C01835=1198.464,47.154,-46.353,-179.303,5.739,148.808
C01836=1198.459,47.403,-46.370,-179.300,5.741,148.808
C01837=1198.454,47.653,-46.386,-179.297,5.741,148.807
C01838=1198.449,47.901,-46.402,-179.295,5.742,148.806
C01839=1198.445,48.152,-46.418,-179.292,5.743,148.806
C01840=1198.439,48.401,-46.434,-179.290,5.743,148.805
C01841=1198.435,48.650,-46.450,-179.287,5.744,148.804
C01842=1198.429,48.900,-46.466,-179.284,5.744,148.804
C01843=1198.425,49.149,-46.482,-179.282,5.745,148.803
C01844=1198.419,49.399,-46.498,-179.280,5.746,148.803
C01845=1198.414,49.647,-46.514,-179.276,5.747,148.802
C01846=1198.410,49.898,-46.530,-179.274,5.748,148.801
C01847=1198.404,50.146,-46.547,-179.272,5.749,148.801
C01848=1198.400,50.396,-46.563,-179.269,5.749,148.800
C01849=1198.395,50.645,-46.579,-179.266,5.750,148.800
C01850=1198.390,50.895,-46.595,-179.264,5.751,148.799
C01851=1198.385,51.144,-46.611,-179.262,5.751,148.798
C01852=1198.380,51.394,-46.627,-179.258,5.753,148.798
C01853=1198.375,51.643,-46.643,-179.256,5.753,148.797
C01854=1198.370,51.893,-46.659,-179.254,5.754,148.797
C01855=1198.365,52.142,-46.676,-179.251,5.754,148.796
C01856=1198.360,52.391,-46.692,-179.248,5.755,148.795
C01857=1198.355,52.641,-46.708,-179.246,5.756,148.795
C01858=1198.351,52.890,-46.725,-179.244,5.756,148.794
C01859=1198.345,53.140,-46.740,-179.240,5.758,148.794
C01860=1198.341,53.389,-46.757,-179.238,5.759,148.793
C01861=1198.336,53.638,-46.773,-179.236,5.759,148.792
C01862=1198.331,53.888,-46.789,-179.233,5.760,148.792
C01863=1198.326,54.138,-46.806,-179.231,5.761,148.791
C01864=1198.321,54.387,-46.823,-179.228,5.761,148.791
C01865=1198.315,54.655,-46.840,-179.225,5.763,148.790
C01866=1198.310,54.924,-46.857,-179.222,5.763,148.789
C01867=1198.305,55.192,-46.875,-179.220,5.764,148.789
C01868=1198.299,55.461,-46.892,-179.216,5.765,148.788
C01869=1198.294,55.710,-46.909,-179.214,5.766,148.788
C01870=1198.290,55.960,-46.926,-179.212,5.766,148.787
C01871=1198.284,56.209,-46.941,-179.209,5.767,148.786
C01872=1198.280,56.459,-46.958,-179.207,5.768,148.786
C01873=1198.275,56.708,-46.974,-179.204,5.768,148.785
C01874=1198.270,56.957,-46.991,-179.201,5.770,148.784
C01875=1198.264,57.207,-47.007,-179.199,5.771,148.784
C01876=1198.260,57.456,-47.024,-179.196,5.771,148.783
C01877=1198.255,57.706,-47.040,-179.194,5.772,148.783
C01878=1198.250,57.955,-47.057,-179.191,5.772,148.782
C01879=1198.244,58.205,-47.073,-179.189,5.773,148.782
C01880=1198.239,58.454,-47.090,-179.186,5.775,148.781
C01881=1198.235,58.703,-47.106,-179.183,5.775,148.780
C01882=1198.230,58.953,-47.123,-179.181,5.776,148.780
C01883=1198.225,59.201,-47.139,-179.178,5.777,148.779
C01884=1198.220,59.452,-47.156,-179.176,5.777,148.779
C01885=1198.215,59.701,-47.172,-179.173,5.778,148.778
C01886=1198.210,59.950,-47.189,-179.170,5.779,148.777
C01887=1198.206,60.200,-47.205,-179.168,5.780,148.777
C01888=1198.200,60.449,-47.222,-179.165,5.781,148.776
C01889=1198.195,60.698,-47.239,-179.163,5.781,148.776
C01890=1198.191,60.948,-47.256,-179.160,5.782,148.775
C01891=1198.185,61.197,-47.273,-179.157,5.784,148.775
C01892=1198.180,61.447,-47.289,-179.155,5.784,148.774
C01893=1198.176,61.696,-47.305,-179.152,5.785,148.773
C01894=1198.171,61.945,-47.321,-179.150,5.786,148.773
C01895=1198.166,62.195,-47.339,-179.147,5.786,148.772
C01896=1198.161,62.444,-47.355,-179.144,5.787,148.771
C01897=1198.156,62.693,-47.372,-179.142,5.788,148.771
C01898=1198.151,62.943,-47.389,-179.139,5.789,148.770
C01899=1198.146,63.192,-47.406,-179.137,5.789,148.770
C01900=1198.141,63.441,-47.422,-179.135,5.790,148.769
C01901=1198.136,63.691,-47.439,-179.131,5.792,148.769
C01902=1198.132,63.941,-47.456,-179.129,5.792,148.768
C01903=1198.126,64.189,-47.472,-179.127,5.793,148.768
C01904=1198.121,64.439,-47.489,-179.124,5.794,148.767
C01905=1198.117,64.689,-47.506,-179.122,5.795,148.766
C01906=1198.112,64.938,-47.523,-179.119,5.796,148.766
C01907=1198.106,65.187,-47.540,-179.116,5.796,148.765
C01908=1198.102,65.437,-47.556,-179.114,5.797,148.765
C01909=1198.097,65.686,-47.574,-179.111,5.798,148.764
C01910=1198.092,65.935,-47.590,-179.109,5.798,148.763
C01911=1198.086,66.185,-47.607,-179.106,5.800,148.763
C01912=1198.082,66.435,-47.624,-179.103,5.801,148.762
C01913=1198.078,66.684,-47.641,-179.101,5.801,148.762
C01914=1198.072,66.933,-47.657,-179.099,5.802,148.761
C01915=1198.067,67.183,-47.674,-179.095,5.804,148.760
C01916=1198.062,67.432,-47.692,-179.093,5.804,148.760
C01917=1198.058,67.681,-47.709,-179.091,5.805,148.759
C01918=1198.052,67.930,-47.726,-179.088,5.806,148.759
C01919=1198.048,68.180,-47.742,-179.085,5.806,148.758
C01920=1198.043,68.429,-47.759,-179.083,5.808,148.758
C01921=1198.038,68.679,-47.776,-179.080,5.808,148.757
C01922=1198.033,68.929,-47.793,-179.078,5.809,148.757
C01923=1198.028,69.177,-47.811,-179.075,5.810,148.756
C01924=1198.023,69.427,-47.827,-179.072,5.811,148.755
C01925=1198.018,69.676,-47.844,-179.070,5.812,148.755
C01926=1198.014,69.926,-47.861,-179.067,5.813,148.754
C01927=1198.008,70.176,-47.878,-179.065,5.813,148.753
C01928=1198.004,70.424,-47.895,-179.062,5.815,148.753
C01929=1197.998,70.674,-47.913,-179.059,5.815,148.752
C01930=1197.994,70.923,-47.929,-179.057,5.816,148.752
C01931=1197.989,71.173,-47.947,-179.054,5.817,148.751
C01932=1197.984,71.422,-47.965,-179.051,5.818,148.751
C01933=1197.979,71.671,-47.981,-179.049,5.819,148.750
C01934=1197.974,71.921,-47.998,-179.046,5.820,148.750
C01935=1197.969,72.170,-48.015,-179.044,5.820,148.749
C01936=1197.964,72.419,-48.033,-179.041,5.822,148.748
C01937=1197.960,72.669,-48.050,-179.038,5.823,148.748
C01938=1197.954,72.919,-48.067,-179.036,5.824,148.747
C01939=1197.949,73.167,-48.084,-179.034,5.824,148.747
C01940=1197.944,73.417,-48.101,-179.030,5.825,148.746
C01941=1197.939,73.666,-48.118,-179.028,5.826,148.746
C01942=1197.935,73.915,-48.136,-179.026,5.827,148.745
C01943=1197.930,74.165,-48.153,-179.023,5.827,148.744
C01944=1197.925,74.415,-48.170,-179.020,5.829,148.744
C01945=1197.920,74.664,-48.188,-179.018,5.830,148.743
C01946=1197.915,74.913,-48.205,-179.016,5.831,148.743
C01947=1197.910,75.162,-48.222,-179.013,5.831,148.742
C01948=1197.905,75.411,-48.239,-179.010,5.833,148.742
C01949=1197.900,75.661,-48.256,-179.008,5.833,148.741
C01950=1197.896,75.910,-48.274,-179.005,5.834,148.740
C01951=1197.891,76.160,-48.291,-179.002,5.836,148.740
C01952=1197.886,76.409,-48.309,-179.000,5.836,148.739
C01953=1197.881,76.659,-48.326,-178.997,5.837,148.739
C01954=1197.876,76.908,-48.344,-178.995,5.838,148.738
C01955=1197.871,77.157,-48.361,-178.992,5.839,148.738
C01956=1197.866,77.406,-48.378,-178.990,5.840,148.737
C01957=1197.861,77.655,-48.395,-178.987,5.841,148.737
C01958=1197.856,77.905,-48.413,-178.984,5.841,148.736
C01959=1197.851,78.154,-48.430,-178.982,5.843,148.735
C01960=1197.847,78.403,-48.448,-178.979,5.843,148.735
C01961=1197.842,78.653,-48.465,-178.977,5.844,148.734
C01962=1197.837,78.902,-48.483,-178.974,5.846,148.734
C01963=1197.831,79.152,-48.500,-178.971,5.846,148.733
C01964=1197.827,79.401,-48.518,-178.969,5.847,148.733
C01965=1197.822,79.651,-48.535,-178.966,5.849,148.732
C01966=1197.817,79.900,-48.553,-178.964,5.850,148.732
C01967=1197.812,80.150,-48.570,-178.961,5.850,148.731
C01968=1197.808,80.399,-48.588,-178.958,5.851,148.730
C01969=1197.802,80.667,-48.606,-178.956,5.852,148.730
C01970=1197.797,80.935,-48.625,-178.953,5.853,148.729
C01971=1197.791,81.204,-48.644,-178.950,5.854,148.729
C01972=1197.786,81.472,-48.664,-178.947,5.855,148.728
C01973=1197.781,81.721,-48.681,-178.944,5.857,148.727
C01974=1197.777,81.971,-48.698,-178.942,5.857,148.727
C01975=1197.772,82.220,-48.716,-178.940,5.858,148.726
C01976=1197.767,82.469,-48.734,-178.936,5.859,148.726
C01977=1197.762,82.719,-48.751,-178.934,5.860,148.725
C01978=1197.757,82.968,-48.769,-178.932,5.861,148.725
C01979=1197.752,83.217,-48.787,-178.928,5.862,148.724
C01980=1197.747,83.467,-48.804,-178.926,5.863,148.724
C01981=1197.743,83.716,-48.822,-178.924,5.864,148.723
C01982=1197.738,83.965,-48.840,-178.921,5.864,148.722
C01983=1197.732,84.215,-48.857,-178.918,5.866,148.722
C01984=1197.728,84.464,-48.875,-178.916,5.867,148.721
C01985=1197.723,84.713,-48.893,-178.914,5.868,148.721
C01986=1197.718,84.962,-48.911,-178.910,5.869,148.720
C01987=1197.713,85.212,-48.928,-178.908,5.870,148.720
C01988=1197.708,85.461,-48.946,-178.906,5.870,148.719
C01989=1197.703,85.710,-48.964,-178.903,5.872,148.719
C01990=1197.699,85.959,-48.982,-178.900,5.873,148.718
C01991=1197.694,86.209,-49.000,-178.898,5.873,148.717
C01992=1197.688,86.458,-49.017,-178.895,5.875,148.717
C01993=1197.683,86.708,-49.035,-178.892,5.876,148.716
C01994=1197.679,86.957,-49.053,-178.890,5.876,148.716
C01995=1197.674,87.207,-49.071,-178.887,5.878,148.715
C01996=1197.669,87.456,-49.089,-178.885,5.879,148.715
C01997=1197.664,87.705,-49.107,-178.882,5.879,148.714
C01998=1197.659,87.955,-49.125,-178.879,5.881,148.713
C01999=1197.654,88.204,-49.143,-178.877,5.882,148.713
C02000=1197.649,88.453,-49.161,-178.874,5.883,148.712
C02001=1197.644,88.702,-49.178,-178.872,5.884,148.712
C02002=1197.640,88.951,-49.196,-178.869,5.884,148.711
C02003=1197.635,89.201,-49.214,-178.866,5.886,148.711
C02004=1197.630,89.451,-49.233,-178.864,5.887,148.710
C02005=1197.625,89.700,-49.251,-178.861,5.888,148.710
C02006=1197.621,89.949,-49.269,-178.858,5.889,148.709
C02007=1197.616,90.198,-49.287,-178.856,5.890,148.709
C02008=1197.611,90.447,-49.305,-178.854,5.891,148.708
C02009=1197.606,90.696,-49.323,-178.850,5.892,148.707
C02010=1197.601,90.946,-49.341,-178.848,5.893,148.707
C02011=1197.596,91.195,-49.359,-178.846,5.893,148.706
C02012=1197.592,91.445,-49.377,-178.843,5.895,148.706
C02013=1197.587,91.694,-49.395,-178.840,5.896,148.705
C02014=1197.582,91.943,-49.413,-178.838,5.898,148.705
C02015=1197.577,92.192,-49.431,-178.835,5.898,148.704
C02016=1197.572,92.441,-49.449,-178.833,5.899,148.704
C02017=1197.567,92.690,-49.467,-178.830,5.900,148.703
C02018=1197.562,92.941,-49.486,-178.827,5.901,148.703
C02019=1197.557,93.190,-49.504,-178.825,5.902,148.702
C02020=1197.552,93.439,-49.522,-178.822,5.904,148.702
C02021=1197.547,93.688,-49.540,-178.820,5.904,148.701
C02022=1197.542,93.937,-49.558,-178.817,5.906,148.701
C02023=1197.538,94.187,-49.576,-178.814,5.906,148.700
C02024=1197.533,94.436,-49.594,-178.812,5.907,148.699
C02025=1197.528,94.686,-49.612,-178.809,5.909,148.699
C02026=1197.523,94.934,-49.631,-178.806,5.909,148.698
C02027=1197.518,95.184,-49.649,-178.804,5.910,148.698
C02028=1197.514,95.434,-49.668,-178.801,5.912,148.697
C02029=1197.509,95.683,-49.686,-178.799,5.913,148.697
C02030=1197.504,95.932,-49.704,-178.796,5.914,148.696
C02031=1197.499,96.181,-49.722,-178.793,5.915,148.696
C02032=1197.494,96.430,-49.741,-178.791,5.915,148.695
C02033=1197.489,96.680,-49.759,-178.788,5.917,148.695
C02034=1197.484,96.929,-49.777,-178.785,5.918,148.694
C02035=1197.479,97.178,-49.795,-178.783,5.920,148.694
C02036=1197.475,97.427,-49.813,-178.780,5.920,148.693
C02037=1197.470,97.677,-49.833,-178.778,5.921,148.693
C02038=1197.465,97.926,-49.851,-178.775,5.922,148.692
C02039=1197.460,98.175,-49.869,-178.773,5.923,148.691
C02040=1197.455,98.424,-49.887,-178.770,5.925,148.691
C02041=1197.450,98.674,-49.906,-178.767,5.926,148.690
C02042=1197.445,98.923,-49.924,-178.765,5.926,148.690
C02043=1197.441,99.172,-49.942,-178.762,5.928,148.689
C02044=1197.436,99.422,-49.961,-178.759,5.929,148.689
C02045=1197.431,99.671,-49.980,-178.757,5.930,148.688
C02046=1197.426,99.920,-49.998,-178.754,5.931,148.688
C02047=1197.421,100.169,-50.017,-178.751,5.933,148.687
C02048=1197.417,100.419,-50.035,-178.749,5.933,148.687
C02049=1197.411,100.668,-50.054,-178.747,5.934,148.686
C02050=1197.407,100.917,-50.072,-178.743,5.936,148.686
C02051=1197.402,101.167,-50.091,-178.741,5.936,148.685
C02052=1197.397,101.416,-50.109,-178.738,5.938,148.685
C02053=1197.392,101.665,-50.128,-178.736,5.939,148.684
C02054=1197.388,101.915,-50.146,-178.733,5.939,148.683
C02055=1197.383,102.163,-50.166,-178.731,5.941,148.683
C02056=1197.378,102.413,-50.184,-178.728,5.942,148.682
C02057=1197.373,102.662,-50.202,-178.725,5.943,148.682
C02058=1197.368,102.911,-50.221,-178.723,5.944,148.681
C02059=1197.363,103.160,-50.239,-178.720,5.946,148.681
C02060=1197.359,103.410,-50.258,-178.717,5.946,148.680
C02061=1197.353,103.659,-50.277,-178.715,5.948,148.680
C02062=1197.349,103.908,-50.296,-178.713,5.949,148.679
C02063=1197.344,104.158,-50.314,-178.710,5.950,148.679
C02064=1197.339,104.407,-50.333,-178.707,5.951,148.678
C02065=1197.335,104.656,-50.351,-178.705,5.952,148.678
C02066=1197.329,104.905,-50.371,-178.702,5.954,148.677
C02067=1197.325,105.154,-50.389,-178.699,5.954,148.677
C02068=1197.320,105.404,-50.408,-178.697,5.956,148.676
C02069=1197.315,105.653,-50.426,-178.694,5.957,148.676
C02070=1197.310,105.902,-50.446,-178.691,5.958,148.675
C02071=1197.305,106.152,-50.464,-178.689,5.959,148.675
C02072=1197.301,106.401,-50.483,-178.687,5.960,148.674
C02073=1197.295,106.670,-50.503,-178.683,5.961,148.674
C02074=1197.290,106.938,-50.524,-178.681,5.963,148.673
C02075=1197.285,107.206,-50.543,-178.678,5.964,148.673
C02076=1197.280,107.475,-50.564,-178.675,5.965,148.672
C02077=1197.274,107.724,-50.583,-178.672,5.967,148.672
C02078=1197.270,107.973,-50.602,-178.670,5.967,148.671
C02079=1197.265,108.222,-50.621,-178.667,5.968,148.670
C02080=1197.260,108.471,-50.639,-178.664,5.970,148.670
C02081=1197.255,108.721,-50.659,-178.662,5.971,148.669
C02082=1197.251,108.970,-50.678,-178.659,5.972,148.669
C02083=1197.246,109.220,-50.697,-178.657,5.973,148.668
C02084=1197.241,109.468,-50.715,-178.654,5.975,148.668
C02085=1197.236,109.718,-50.735,-178.652,5.975,148.667
C02086=1197.232,109.966,-50.754,-178.649,5.977,148.667
C02087=1197.227,110.217,-50.773,-178.646,5.978,148.666
C02088=1197.222,110.465,-50.791,-178.644,5.979,148.666
C02089=1197.217,110.715,-50.811,-178.641,5.980,148.665
C02090=1197.212,110.964,-50.829,-178.638,5.982,148.665
C02091=1197.208,111.213,-50.848,-178.636,5.983,148.664
C02092=1197.202,111.462,-50.868,-178.633,5.984,148.664
C02093=1197.198,111.712,-50.887,-178.631,5.985,148.663
C02094=1197.193,111.960,-50.906,-178.628,5.986,148.663
C02095=1197.189,112.210,-50.924,-178.625,5.987,148.662
C02096=1197.183,112.459,-50.944,-178.622,5.989,148.662
C02097=1197.179,112.709,-50.963,-178.620,5.990,148.661
C02098=1197.174,112.957,-50.982,-178.617,5.991,148.661
C02099=1197.169,113.207,-51.002,-178.615,5.992,148.660
C02100=1197.164,113.456,-51.020,-178.612,5.994,148.660
C02101=1197.160,113.706,-51.039,-178.610,5.994,148.659
C02102=1197.154,113.954,-51.059,-178.607,5.996,148.659
C02103=1197.149,114.204,-51.078,-178.604,5.997,148.658
C02104=1197.145,114.453,-51.097,-178.601,5.998,148.658
C02105=1197.140,114.702,-51.117,-178.599,5.999,148.657
C02106=1197.135,114.951,-51.136,-178.596,6.001,148.657
C02107=1197.131,115.200,-51.155,-178.594,6.002,148.656
C02108=1197.125,115.449,-51.174,-178.591,6.003,148.656
C02109=1197.120,115.699,-51.193,-178.589,6.004,148.655
C02110=1197.116,115.949,-51.212,-178.586,6.006,148.655
C02111=1197.111,116.197,-51.232,-178.583,6.006,148.654
C02112=1197.106,116.447,-51.251,-178.581,6.008,148.654
C02113=1197.101,116.696,-51.271,-178.578,6.009,148.653
C02114=1197.097,116.945,-51.290,-178.575,6.010,148.653
C02115=1197.092,117.194,-51.309,-178.573,6.011,148.652
C02116=1197.087,117.444,-51.329,-178.570,6.013,148.652
C02117=1197.082,117.693,-51.348,-178.568,6.014,148.651
C02118=1197.077,117.942,-51.367,-178.565,6.015,148.651
C02119=1197.073,118.191,-51.387,-178.563,6.016,148.650
C02120=1197.067,118.440,-51.406,-178.560,6.017,148.650
C02121=1197.063,118.690,-51.426,-178.557,6.018,148.649
C02122=1197.058,118.939,-51.446,-178.555,6.020,148.649
C02123=1197.054,119.187,-51.465,-178.552,6.022,148.648
C02124=1197.049,119.437,-51.484,-178.549,6.022,148.648
C02125=1197.044,119.686,-51.504,-178.546,6.024,148.647
C02126=1197.039,119.935,-51.523,-178.544,6.025,148.647
C02127=1197.034,120.185,-51.543,-178.541,6.027,148.646
C02128=1197.030,120.434,-51.562,-178.539,6.027,148.646
C02129=1197.025,120.683,-51.581,-178.536,6.029,148.645
C02130=1197.020,120.933,-51.601,-178.534,6.030,148.645
C02131=1197.015,121.181,-51.620,-178.531,6.031,148.644
C02132=1197.010,121.430,-51.641,-178.529,6.032,148.644
C02133=1197.005,121.680,-51.660,-178.525,6.034,148.643
C02134=1197.000,121.929,-51.680,-178.523,6.035,148.643
C02135=1196.996,122.178,-51.699,-178.521,6.036,148.643
C02136=1196.991,122.428,-51.718,-178.517,6.038,148.642
C02137=1196.987,122.677,-51.739,-178.515,6.039,148.641
C02138=1196.982,122.925,-51.758,-178.513,6.040,148.641
C02139=1196.977,123.175,-51.778,-178.510,6.041,148.640
C02140=1196.972,123.425,-51.797,-178.507,6.043,148.640
C02141=1196.967,123.673,-51.817,-178.505,6.043,148.639
C02142=1196.962,123.922,-51.837,-178.502,6.045,148.639
C02143=1196.958,124.172,-51.857,-178.499,6.047,148.639
C02144=1196.952,124.421,-51.876,-178.497,6.048,148.638
C02145=1196.948,124.670,-51.896,-178.494,6.049,148.638
C02146=1196.944,124.919,-51.915,-178.492,6.050,148.637
C02147=1196.939,125.169,-51.935,-178.489,6.052,148.637
C02148=1196.934,125.417,-51.955,-178.487,6.053,148.636
C02149=1196.929,125.666,-51.975,-178.484,6.054,148.636
C02150=1196.924,125.916,-51.994,-178.481,6.056,148.635
C02151=1196.920,126.165,-52.015,-178.479,6.057,148.635
C02152=1196.915,126.414,-52.034,-178.475,6.058,148.634
C02153=1196.910,126.663,-52.054,-178.473,6.059,148.634
C02154=1196.906,126.912,-52.074,-178.471,6.061,148.633
C02155=1196.901,127.162,-52.094,-178.467,6.062,148.633
C02156=1196.896,127.410,-52.114,-178.465,6.063,148.632
C02157=1196.891,127.660,-52.133,-178.463,6.065,148.632
C02158=1196.886,127.909,-52.153,-178.460,6.066,148.631
C02159=1196.882,128.158,-52.173,-178.457,6.067,148.631
C02160=1196.877,128.408,-52.193,-178.455,6.068,148.630
C02161=1196.872,128.656,-52.213,-178.452,6.070,148.630
C02162=1196.867,128.906,-52.233,-178.449,6.071,148.629
C02163=1196.862,129.155,-52.254,-178.447,6.072,148.629
C02164=1196.857,129.404,-52.273,-178.444,6.074,148.628
C02165=1196.853,129.653,-52.294,-178.442,6.075,148.628
C02166=1196.848,129.902,-52.313,-178.439,6.077,148.628
C02167=1196.843,130.151,-52.333,-178.436,6.078,148.627
C02168=1196.838,130.401,-52.353,-178.434,6.079,148.627
C02169=1196.834,130.650,-52.373,-178.431,6.081,148.626
C02170=1196.829,130.899,-52.393,-178.429,6.081,148.626
C02171=1196.824,131.147,-52.413,-178.426,6.083,148.625
C02172=1196.819,131.397,-52.433,-178.423,6.085,148.625
C02173=1196.814,131.646,-52.454,-178.421,6.085,148.624
C02174=1196.810,131.896,-52.473,-178.418,6.087,148.624
C02175=1196.805,132.145,-52.494,-178.415,6.089,148.623
C02176=1196.801,132.394,-52.514,-178.413,6.090,148.623
C02177=1196.795,132.663,-52.536,-178.410,6.091,148.622
C02178=1196.790,132.931,-52.557,-178.407,6.093,148.622
C02179=1196.785,133.200,-52.579,-178.404,6.094,148.621
C02180=1196.780,133.468,-52.600,-178.401,6.096,148.621
C02181=1196.775,133.718,-52.621,-178.399,6.097,148.620
C02182=1196.770,133.967,-52.642,-178.396,6.099,148.620
C02183=1196.765,134.216,-52.661,-178.394,6.100,148.620
C02184=1196.760,134.464,-52.681,-178.391,6.101,148.619
C02185=1196.756,134.713,-52.702,-178.388,6.103,148.619
C02186=1196.751,134.963,-52.722,-178.386,6.104,148.618
C02187=1196.746,135.212,-52.742,-178.383,6.105,148.618
C02188=1196.742,135.461,-52.763,-178.380,6.107,148.617
C02189=1196.737,135.711,-52.782,-178.378,6.108,148.617
C02190=1196.732,135.960,-52.803,-178.375,6.109,148.616
C02191=1196.727,136.209,-52.824,-178.372,6.111,148.616
C02192=1196.723,136.458,-52.844,-178.370,6.112,148.615
C02193=1196.718,136.707,-52.864,-178.367,6.114,148.615
C02194=1196.713,136.957,-52.885,-178.365,6.114,148.614
C02195=1196.708,137.206,-52.905,-178.362,6.116,148.614
C02196=1196.703,137.454,-52.925,-178.359,6.118,148.614
C02197=1196.698,137.703,-52.946,-178.357,6.119,148.613
C02198=1196.694,137.952,-52.966,-178.354,6.120,148.613
C02199=1196.689,138.202,-52.986,-178.352,6.122,148.612
C02200=1196.684,138.451,-53.007,-178.349,6.123,148.612
C02201=1196.679,138.700,-53.027,-178.346,6.124,148.611
C02202=1196.675,138.949,-53.048,-178.344,6.126,148.611
C02203=1196.670,139.198,-53.069,-178.341,6.127,148.610
C02204=1196.665,139.447,-53.089,-178.338,6.129,148.610
C02205=1196.661,139.696,-53.109,-178.336,6.130,148.609
C02206=1196.656,139.945,-53.130,-178.333,6.131,148.609
C02207=1196.651,140.195,-53.150,-178.331,6.133,148.609
C02208=1196.647,140.444,-53.170,-178.328,6.135,148.608
C02209=1196.641,140.693,-53.191,-178.325,6.135,148.608
C02210=1196.637,140.942,-53.212,-178.323,6.137,148.607
C02211=1196.632,141.191,-53.233,-178.320,6.139,148.607
C02212=1196.627,141.440,-53.253,-178.318,6.140,148.606
C02213=1196.623,141.689,-53.273,-178.315,6.141,148.606
C02214=1196.618,141.938,-53.294,-178.312,6.143,148.605
C02215=1196.613,142.187,-53.315,-178.310,6.144,148.605
C02216=1196.608,142.437,-53.336,-178.307,6.146,148.604
C02217=1196.604,142.686,-53.356,-178.304,6.147,148.604
C02218=1196.599,142.935,-53.377,-178.301,6.149,148.604
C02219=1196.594,143.184,-53.397,-178.299,6.150,148.603
C02220=1196.590,143.433,-53.418,-178.296,6.151,148.603
C02221=1196.585,143.683,-53.439,-178.294,6.153,148.602
C02222=1196.581,143.932,-53.459,-178.291,6.154,148.602
C02223=1196.576,144.180,-53.481,-178.288,6.156,148.601
C02224=1196.571,144.429,-53.502,-178.286,6.157,148.601
C02225=1196.566,144.678,-53.522,-178.283,6.158,148.601
C02226=1196.562,144.927,-53.543,-178.281,6.160,148.600
C02227=1196.557,145.177,-53.564,-178.278,6.162,148.600
C02228=1196.552,145.426,-53.584,-178.275,6.163,148.599
C02229=1196.547,145.675,-53.605,-178.273,6.164,148.599
C02230=1196.543,145.924,-53.626,-178.270,6.166,148.598
C02231=1196.538,146.172,-53.647,-178.267,6.168,148.598
C02232=1196.533,146.421,-53.668,-178.265,6.168,148.597
C02233=1196.529,146.671,-53.689,-178.262,6.170,148.597
C02234=1196.523,146.921,-53.710,-178.259,6.172,148.597
C02235=1196.519,147.170,-53.730,-178.257,6.173,148.596
C02236=1196.514,147.418,-53.752,-178.254,6.174,148.596
C02237=1196.510,147.667,-53.772,-178.252,6.176,148.595
C02238=1196.505,147.916,-53.793,-178.249,6.178,148.595
C02239=1196.499,148.166,-53.814,-178.247,6.179,148.594
C02240=1196.495,148.415,-53.835,-178.244,6.181,148.594
C02241=1196.491,148.664,-53.857,-178.241,6.182,148.593
C02242=1196.486,148.913,-53.877,-178.238,6.184,148.593
C02243=1196.481,149.162,-53.898,-178.236,6.185,148.593
C02244=1196.476,149.411,-53.920,-178.233,6.187,148.592
C02245=1196.472,149.660,-53.940,-178.230,6.188,148.592
C02246=1196.467,149.909,-53.961,-178.228,6.189,148.591
C02247=1196.462,150.158,-53.983,-178.225,6.191,148.591
C02248=1196.458,150.407,-54.003,-178.223,6.193,148.591
C02249=1196.453,150.657,-54.024,-178.220,6.194,148.590
C02250=1196.448,150.905,-54.046,-178.217,6.195,148.590
C02251=1196.443,151.154,-54.066,-178.215,6.197,148.589
C02252=1196.438,151.403,-54.087,-178.212,6.199,148.589
C02253=1196.434,151.653,-54.109,-178.209,6.200,148.588
C02254=1196.430,151.902,-54.130,-178.207,6.201,148.588
C02255=1196.425,152.150,-54.152,-178.204,6.203,148.587
C02256=1196.419,152.400,-54.173,-178.201,6.205,148.587
C02257=1196.414,152.649,-54.193,-178.199,6.206,148.587
C02258=1196.411,152.898,-54.215,-178.197,6.207,148.586
C02259=1196.406,153.147,-54.236,-178.194,6.209,148.586
C02260=1196.401,153.396,-54.258,-178.191,6.210,148.585
C02261=1196.396,153.645,-54.279,-178.188,6.212,148.585
C02262=1196.392,153.894,-54.300,-178.186,6.213,148.585
C02263=1196.387,154.143,-54.321,-178.183,6.215,148.584
C02264=1196.382,154.392,-54.343,-178.181,6.217,148.584
C02265=1196.377,154.641,-54.364,-178.178,6.219,148.583
C02266=1196.373,154.890,-54.385,-178.175,6.220,148.583
C02267=1196.368,155.140,-54.406,-178.173,6.221,148.582
C02268=1196.363,155.388,-54.428,-178.170,6.223,148.582
C02269=1196.358,155.637,-54.449,-178.167,6.225,148.582
C02270=1196.354,155.887,-54.471,-178.165,6.226,148.581
C02271=1196.350,156.135,-54.492,-178.162,6.227,148.581
C02272=1196.344,156.384,-54.513,-178.159,6.229,148.580
C02273=1196.340,156.633,-54.534,-178.157,6.230,148.580
C02274=1196.335,156.883,-54.556,-178.154,6.232,148.580
C02275=1196.330,157.132,-54.577,-178.152,6.233,148.579
C02276=1196.325,157.380,-54.599,-178.149,6.235,148.579
C02277=1196.321,157.630,-54.621,-178.147,6.237,148.578
C02278=1196.317,157.879,-54.642,-178.143,6.238,148.578
C02279=1196.312,158.127,-54.663,-178.141,6.240,148.577
C02280=1196.307,158.377,-54.685,-178.139,6.241,148.577
C02281=1196.302,158.646,-54.709,-178.136,6.243,148.577
C02282=1196.297,158.915,-54.731,-178.133,6.244,148.576
C02283=1196.291,159.184,-54.754,-178.130,6.246,148.576
C02284=1196.286,159.453,-54.777,-178.128,6.248,148.575
C02285=1196.282,159.702,-54.799,-178.125,6.250,148.575
C02286=1196.277,159.951,-54.821,-178.122,6.251,148.574
C02287=1196.272,160.199,-54.843,-178.119,6.253,148.574
C02288=1196.268,160.449,-54.864,-178.116,6.255,148.574
C02289=1196.263,160.698,-54.886,-178.114,6.256,148.573
C02290=1196.259,160.947,-54.908,-178.112,6.257,148.573
C02291=1196.254,161.196,-54.929,-178.109,6.259,148.573
C02292=1196.249,161.445,-54.951,-178.106,6.261,148.572
C02293=1196.244,161.694,-54.972,-178.103,6.262,148.572
C02294=1196.240,161.943,-54.994,-178.100,6.264,148.571
C02295=1196.235,162.192,-55.016,-178.098,6.265,148.571
C02296=1196.230,162.441,-55.038,-178.096,6.267,148.570
C02297=1196.226,162.690,-55.059,-178.093,6.269,148.570
C02298=1196.221,162.939,-55.082,-178.090,6.270,148.570
C02299=1196.216,163.188,-55.102,-178.088,6.272,148.569
C02300=1196.211,163.437,-55.124,-178.085,6.273,148.569
C02301=1196.207,163.686,-55.146,-178.082,6.275,148.568
C02302=1196.202,163.935,-55.168,-178.080,6.276,148.568
C02303=1196.198,164.184,-55.190,-178.077,6.278,148.568
C02304=1196.193,164.433,-55.212,-178.074,6.280,148.567
C02305=1196.189,164.682,-55.234,-178.072,6.282,148.567
C02306=1196.184,164.931,-55.255,-178.069,6.283,148.566
C02307=1196.179,165.180,-55.277,-178.067,6.285,148.566
C02308=1196.175,165.429,-55.299,-178.064,6.286,148.566
C02309=1196.169,165.678,-55.321,-178.061,6.288,148.565
C02310=1196.165,165.927,-55.343,-178.058,6.290,148.565
C02311=1196.160,166.176,-55.365,-178.056,6.291,148.564
C02312=1196.156,166.425,-55.387,-178.053,6.293,148.564
C02313=1196.151,166.674,-55.409,-178.051,6.294,148.564
C02314=1196.146,166.923,-55.431,-178.048,6.296,148.563
C02315=1196.142,167.172,-55.453,-178.046,6.298,148.563
C02316=1196.137,167.421,-55.475,-178.043,6.300,148.563
C02317=1196.132,167.670,-55.497,-178.040,6.301,148.562
C02318=1196.127,167.919,-55.519,-178.038,6.303,148.562
C02319=1196.123,168.168,-55.541,-178.035,6.304,148.561
C02320=1196.118,168.417,-55.563,-178.032,6.306,148.561
C02321=1196.113,168.666,-55.584,-178.030,6.307,148.560
C02322=1196.110,168.915,-55.607,-178.027,6.309,148.560
C02323=1196.104,169.164,-55.629,-178.024,6.311,148.560
C02324=1196.100,169.413,-55.651,-178.022,6.313,148.559
C02325=1196.095,169.662,-55.673,-178.019,6.315,148.559
C02326=1196.091,169.911,-55.695,-178.017,6.315,148.559
C02327=1196.085,170.160,-55.717,-178.014,6.317,148.558
C02328=1196.081,170.409,-55.740,-178.011,6.319,148.558
C02329=1196.076,170.657,-55.762,-178.009,6.321,148.558
C02330=1196.072,170.907,-55.784,-178.006,6.323,148.557
C02331=1196.066,171.156,-55.806,-178.003,6.324,148.557
C02332=1196.062,171.405,-55.828,-178.000,6.326,148.556
C02333=1196.058,171.654,-55.851,-177.998,6.328,148.556
C02334=1196.053,171.902,-55.873,-177.996,6.329,148.555
C02335=1196.048,172.152,-55.895,-177.993,6.330,148.555
C02336=1196.043,172.401,-55.917,-177.990,6.332,148.555
C02337=1196.039,172.649,-55.940,-177.988,6.334,148.554
C02338=1196.034,172.898,-55.962,-177.985,6.336,148.554
C02339=1196.029,173.148,-55.984,-177.982,6.338,148.554
C02340=1196.025,173.396,-56.007,-177.980,6.339,148.553
C02341=1196.020,173.645,-56.029,-177.977,6.341,148.553
C02342=1196.016,173.895,-56.051,-177.974,6.343,148.553
C02343=1196.011,174.143,-56.074,-177.971,6.345,148.552
C02344=1196.006,174.392,-56.096,-177.969,6.346,148.552
C02345=1196.002,174.642,-56.118,-177.967,6.348,148.551
C02346=1195.997,174.890,-56.141,-177.964,6.349,148.551
C02347=1195.992,175.139,-56.163,-177.961,6.351,148.551
C02348=1195.988,175.387,-56.186,-177.959,6.353,148.550
C02349=1195.983,175.637,-56.208,-177.956,6.355,148.550
C02350=1195.978,175.886,-56.230,-177.953,6.356,148.549
C02351=1195.974,176.134,-56.253,-177.950,6.358,148.549
C02352=1195.969,176.384,-56.275,-177.948,6.360,148.549
C02353=1195.965,176.633,-56.298,-177.945,6.362,148.548
C02354=1195.960,176.881,-56.320,-177.943,6.363,148.548
C02355=1195.955,177.130,-56.343,-177.940,6.364,148.548
C02356=1195.951,177.380,-56.365,-177.937,6.366,148.547
C02357=1195.946,177.628,-56.388,-177.935,6.368,148.547
C02358=1195.941,177.877,-56.410,-177.932,6.370,148.547
C02359=1195.937,178.126,-56.434,-177.929,6.372,148.546
C02360=1195.932,178.375,-56.455,-177.927,6.373,148.546
C02361=1195.927,178.624,-56.479,-177.924,6.375,148.545
C02362=1195.923,178.874,-56.501,-177.921,6.377,148.545
C02363=1195.918,179.122,-56.524,-177.919,6.379,148.545
C02364=1195.913,179.371,-56.546,-177.916,6.381,148.544
C02365=1195.909,179.620,-56.569,-177.913,6.382,148.544
C02366=1195.905,179.869,-56.592,-177.911,6.384,148.544
C02367=1195.899,180.118,-56.614,-177.908,6.386,148.543
C02368=1195.895,180.367,-56.637,-177.906,6.387,148.543
C02369=1195.890,180.616,-56.660,-177.903,6.389,148.543
C02370=1195.885,180.864,-56.682,-177.901,6.391,148.542
C02371=1195.881,181.113,-56.705,-177.898,6.392,148.542
C02372=1195.876,181.363,-56.727,-177.895,6.394,148.541
C02373=1195.872,181.612,-56.751,-177.893,6.396,148.541
C02374=1195.867,181.860,-56.773,-177.890,6.398,148.541
C02375=1195.862,182.109,-56.796,-177.887,6.400,148.540
C02376=1195.858,182.358,-56.819,-177.885,6.401,148.540
C02377=1195.854,182.607,-56.842,-177.882,6.403,148.540
C02378=1195.848,182.855,-56.865,-177.879,6.405,148.539
C02379=1195.844,183.105,-56.887,-177.877,6.407,148.539
C02380=1195.839,183.354,-56.910,-177.874,6.409,148.539
C02381=1195.835,183.603,-56.934,-177.871,6.410,148.538
C02382=1195.831,183.852,-56.957,-177.869,6.412,148.538
C02383=1195.825,184.101,-56.979,-177.866,6.414,148.538
C02384=1195.821,184.349,-57.002,-177.863,6.416,148.537
C02385=1195.816,184.619,-57.027,-177.861,6.418,148.537
C02386=1195.810,184.889,-57.052,-177.858,6.419,148.537
C02387=1195.806,185.158,-57.076,-177.855,6.421,148.536
C02388=1195.801,185.427,-57.102,-177.852,6.424,148.536
C02389=1195.796,185.677,-57.124,-177.850,6.426,148.535
C02390=1195.792,185.926,-57.147,-177.847,6.427,148.535
C02391=1195.787,186.175,-57.171,-177.845,6.428,148.535
C02392=1195.782,186.424,-57.194,-177.842,6.430,148.534
C02393=1195.778,186.672,-57.216,-177.839,6.432,148.534
C02394=1195.773,186.921,-57.240,-177.837,6.434,148.534
C02395=1195.769,187.170,-57.263,-177.834,6.436,148.533
C02396=1195.764,187.419,-57.286,-177.831,6.437,148.533
C02397=1195.760,187.668,-57.309,-177.829,6.439,148.533
C02398=1195.755,187.917,-57.333,-177.826,6.441,148.532
C02399=1195.750,188.165,-57.356,-177.823,6.443,148.532
C02400=1195.745,188.414,-57.379,-177.821,6.445,148.532
C02401=1195.741,188.663,-57.402,-177.818,6.446,148.531
C02402=1195.736,188.912,-57.425,-177.815,6.448,148.531
C02403=1195.732,189.161,-57.448,-177.813,6.450,148.531
C02404=1195.727,189.410,-57.472,-177.810,6.452,148.530
C02405=1195.722,189.659,-57.495,-177.807,6.454,148.530
C02406=1195.718,189.908,-57.518,-177.805,6.455,148.529
C02407=1195.714,190.157,-57.541,-177.802,6.457,148.529
C02408=1195.708,190.405,-57.564,-177.800,6.459,148.529
C02409=1195.704,190.654,-57.588,-177.797,6.461,148.528
C02410=1195.699,190.903,-57.611,-177.795,6.463,148.528
C02411=1195.694,191.152,-57.634,-177.792,6.465,148.528
C02412=1195.690,191.401,-57.657,-177.789,6.467,148.528
C02413=1195.686,191.650,-57.680,-177.787,6.468,148.527
C02414=1195.681,191.899,-57.704,-177.784,6.470,148.527
C02415=1195.676,192.148,-57.727,-177.781,6.472,148.527
C02416=1195.672,192.396,-57.751,-177.779,6.474,148.526
C02417=1195.667,192.645,-57.775,-177.776,6.476,148.526
C02418=1195.662,192.894,-57.798,-177.773,6.478,148.526
C02419=1195.658,193.143,-57.821,-177.770,6.480,148.525
C02420=1195.653,193.392,-57.845,-177.768,6.482,148.525
C02421=1195.649,193.641,-57.868,-177.765,6.484,148.524
C02422=1195.645,193.890,-57.891,-177.762,6.485,148.524
C02423=1195.640,194.139,-57.915,-177.760,6.487,148.524
C02424=1195.635,194.388,-57.938,-177.757,6.489,148.524
C02425=1195.630,194.636,-57.961,-177.755,6.491,148.523
C02426=1195.626,194.884,-57.985,-177.752,6.493,148.523
C02427=1195.621,195.133,-58.009,-177.749,6.495,148.523
C02428=1195.616,195.382,-58.032,-177.747,6.497,148.522
C02429=1195.612,195.631,-58.056,-177.744,6.498,148.522
C02430=1195.607,195.880,-58.079,-177.741,6.500,148.522
C02431=1195.602,196.129,-58.103,-177.739,6.502,148.521
C02432=1195.599,196.378,-58.127,-177.736,6.504,148.521
C02433=1195.594,196.627,-58.151,-177.733,6.506,148.520
C02434=1195.589,196.876,-58.174,-177.731,6.508,148.520
C02435=1195.585,197.125,-58.198,-177.729,6.510,148.520
C02436=1195.580,197.374,-58.221,-177.726,6.511,148.520
C02437=1195.575,197.623,-58.245,-177.723,6.513,148.519
C02438=1195.571,197.871,-58.269,-177.721,6.515,148.519
C02439=1195.566,198.120,-58.292,-177.718,6.517,148.519
C02440=1195.562,198.368,-58.316,-177.715,6.519,148.518
C02441=1195.557,198.617,-58.340,-177.712,6.521,148.518
C02442=1195.552,198.867,-58.364,-177.709,6.523,148.518
C02443=1195.547,199.115,-58.388,-177.707,6.525,148.518
C02444=1195.543,199.364,-58.411,-177.705,6.527,148.517
C02445=1195.538,199.613,-58.435,-177.702,6.529,148.517
C02446=1195.534,199.862,-58.458,-177.699,6.531,148.516
C02447=1195.529,200.110,-58.482,-177.697,6.533,148.516
C02448=1195.525,200.359,-58.506,-177.694,6.534,148.516
C02449=1195.521,200.608,-58.530,-177.691,6.536,148.515
C02450=1195.516,200.857,-58.554,-177.689,6.538,148.515
C02451=1195.511,201.106,-58.578,-177.686,6.540,148.515
C02452=1195.506,201.355,-58.602,-177.684,6.542,148.515
C02453=1195.502,201.603,-58.626,-177.681,6.544,148.514
C02454=1195.497,201.852,-58.650,-177.679,6.546,148.514
C02455=1195.493,202.101,-58.673,-177.675,6.548,148.514
C02456=1195.488,202.349,-58.697,-177.673,6.550,148.513
C02457=1195.483,202.599,-58.722,-177.670,6.552,148.513
C02458=1195.479,202.848,-58.746,-177.668,6.554,148.513
C02459=1195.475,203.096,-58.770,-177.665,6.556,148.512
C02460=1195.470,203.345,-58.793,-177.662,6.558,148.512
C02461=1195.466,203.594,-58.817,-177.660,6.559,148.512
C02462=1195.460,203.842,-58.842,-177.657,6.561,148.511
C02463=1195.456,204.091,-58.865,-177.655,6.563,148.511
C02464=1195.452,204.340,-58.890,-177.652,6.565,148.511
C02465=1195.448,204.589,-58.914,-177.649,6.568,148.511
C02466=1195.442,204.838,-58.938,-177.646,6.570,148.510
C02467=1195.438,205.087,-58.962,-177.644,6.571,148.510
C02468=1195.433,205.335,-58.986,-177.641,6.573,148.510
C02469=1195.430,205.584,-59.010,-177.639,6.575,148.509
C02470=1195.424,205.834,-59.034,-177.636,6.577,148.509
C02471=1195.420,206.082,-59.058,-177.634,6.579,148.509
C02472=1195.415,206.330,-59.082,-177.631,6.581,148.508
C02473=1195.410,206.579,-59.107,-177.628,6.583,148.508
C02474=1195.406,206.829,-59.131,-177.625,6.585,148.508
C02475=1195.402,207.077,-59.155,-177.623,6.587,148.508
C02476=1195.397,207.326,-59.179,-177.620,6.589,148.507
C02477=1195.392,207.574,-59.204,-177.618,6.591,148.507
C02478=1195.388,207.823,-59.228,-177.615,6.593,148.507
C02479=1195.383,208.072,-59.253,-177.612,6.595,148.506
C02480=1195.379,208.321,-59.276,-177.610,6.597,148.506
C02481=1195.374,208.570,-59.300,-177.607,6.598,148.506
C02482=1195.369,208.818,-59.325,-177.604,6.601,148.506
C02483=1195.365,209.067,-59.349,-177.602,6.603,148.505
C02484=1195.360,209.316,-59.374,-177.599,6.605,148.505
C02485=1195.356,209.565,-59.398,-177.596,6.607,148.505
C02486=1195.351,209.813,-59.422,-177.594,6.609,148.504
C02487=1195.347,210.062,-59.447,-177.592,6.611,148.504
C02488=1195.342,210.311,-59.471,-177.589,6.613,148.504
C02489=1195.337,210.581,-59.498,-177.586,6.615,148.503
C02490=1195.332,210.852,-59.524,-177.583,6.617,148.503
C02491=1195.327,211.123,-59.551,-177.580,6.620,148.503
C02492=1195.322,211.393,-59.578,-177.577,6.621,148.503
C02493=1195.318,211.641,-59.602,-177.575,6.623,148.502
C02494=1195.313,211.891,-59.627,-177.572,6.625,148.502
C02495=1195.309,212.139,-59.651,-177.570,6.627,148.502
C02496=1195.304,212.388,-59.675,-177.567,6.630,148.501
C02497=1195.300,212.637,-59.700,-177.564,6.632,148.501
C02498=1195.295,212.885,-59.724,-177.561,6.634,148.501
C02499=1195.290,213.134,-59.749,-177.559,6.635,148.500
C02500=1195.286,213.383,-59.774,-177.556,6.638,148.500
C02501=1195.282,213.631,-59.799,-177.554,6.639,148.500
C02502=1195.277,213.880,-59.823,-177.551,6.642,148.500
C02503=1195.273,214.129,-59.848,-177.548,6.644,148.499
C02504=1195.268,214.378,-59.872,-177.546,6.646,148.499
C02505=1195.263,214.626,-59.896,-177.543,6.648,148.499
C02506=1195.259,214.876,-59.921,-177.540,6.650,148.499
C02507=1195.255,215.123,-59.946,-177.538,6.651,148.498
C02508=1195.249,215.372,-59.971,-177.535,6.654,148.498
C02509=1195.245,215.622,-59.996,-177.532,6.656,148.498
C02510=1195.241,215.870,-60.020,-177.530,6.658,148.497
C02511=1195.236,216.119,-60.045,-177.527,6.660,148.497
C02512=1195.232,216.367,-60.070,-177.524,6.662,148.497
C02513=1195.227,216.616,-60.094,-177.522,6.665,148.497
C02514=1195.222,216.865,-60.119,-177.519,6.666,148.496
C02515=1195.218,217.114,-60.144,-177.516,6.668,148.496
C02516=1195.214,217.363,-60.169,-177.514,6.670,148.496
C02517=1195.209,217.611,-60.193,-177.512,6.672,148.496
C02518=1195.204,217.860,-60.218,-177.509,6.674,148.495
C02519=1195.200,218.109,-60.244,-177.506,6.677,148.495
C02520=1195.196,218.357,-60.268,-177.503,6.679,148.495
C02521=1195.191,218.606,-60.293,-177.501,6.681,148.494
C02522=1195.186,218.855,-60.318,-177.498,6.683,148.494
C02523=1195.182,219.104,-60.343,-177.496,6.684,148.494
C02524=1195.177,219.352,-60.367,-177.492,6.687,148.494
C02525=1195.173,219.601,-60.393,-177.490,6.689,148.493
C02526=1195.168,219.850,-60.418,-177.488,6.691,148.493
C02527=1195.164,220.098,-60.443,-177.485,6.693,148.493
C02528=1195.159,220.347,-60.468,-177.483,6.695,148.493
C02529=1195.154,220.595,-60.493,-177.480,6.698,148.492
C02530=1195.150,220.845,-60.518,-177.477,6.699,148.492
C02531=1195.146,221.093,-60.542,-177.474,6.701,148.492
C02532=1195.141,221.342,-60.568,-177.472,6.703,148.492
C02533=1195.136,221.591,-60.593,-177.469,6.705,148.491
C02534=1195.132,221.839,-60.618,-177.466,6.708,148.491
C02535=1195.128,222.088,-60.642,-177.464,6.710,148.491
C02536=1195.123,222.337,-60.668,-177.461,6.712,148.490
C02537=1195.118,222.585,-60.693,-177.459,6.714,148.490
C02538=1195.114,222.834,-60.719,-177.456,6.716,148.490
C02539=1195.110,223.083,-60.744,-177.453,6.719,148.490
C02540=1195.105,223.331,-60.768,-177.451,6.720,148.489
C02541=1195.101,223.580,-60.794,-177.448,6.722,148.489
C02542=1195.096,223.829,-60.819,-177.446,6.724,148.489
C02543=1195.092,224.078,-60.845,-177.443,6.727,148.489
C02544=1195.087,224.326,-60.869,-177.440,6.729,148.488
C02545=1195.082,224.575,-60.895,-177.438,6.731,148.488
C02546=1195.078,224.823,-60.920,-177.435,6.733,148.488
C02547=1195.074,225.072,-60.945,-177.432,6.735,148.488
C02548=1195.069,225.321,-60.970,-177.430,6.738,148.488
C02549=1195.065,225.569,-60.996,-177.427,6.739,148.487
C02550=1195.060,225.819,-61.021,-177.425,6.741,148.487
C02551=1195.055,226.067,-61.046,-177.422,6.743,148.487
C02552=1195.051,226.316,-61.072,-177.419,6.746,148.486
C02553=1195.046,226.564,-61.097,-177.417,6.748,148.486
C02554=1195.042,226.813,-61.123,-177.414,6.750,148.486
C02555=1195.038,227.062,-61.148,-177.412,6.752,148.486
C02556=1195.033,227.310,-61.174,-177.409,6.755,148.485
C02557=1195.028,227.560,-61.199,-177.406,6.757,148.485
C02558=1195.023,227.808,-61.224,-177.404,6.758,148.485
C02559=1195.019,228.056,-61.250,-177.401,6.760,148.485
C02560=1195.015,228.305,-61.276,-177.398,6.763,148.485
C02561=1195.010,228.553,-61.301,-177.396,6.765,148.484
C02562=1195.006,228.803,-61.326,-177.393,6.767,148.484
C02563=1195.001,229.052,-61.352,-177.391,6.769,148.484
C02564=1194.997,229.300,-61.377,-177.388,6.772,148.484
C02565=1194.992,229.548,-61.403,-177.385,6.774,148.483
C02566=1194.987,229.797,-61.428,-177.383,6.776,148.483
C02567=1194.983,230.045,-61.454,-177.380,6.778,148.483
C02568=1194.979,230.294,-61.480,-177.378,6.781,148.483
C02569=1194.974,230.543,-61.504,-177.375,6.782,148.482
C02570=1194.970,230.792,-61.530,-177.372,6.784,148.482
C02571=1194.965,231.041,-61.556,-177.370,6.786,148.482
C02572=1194.961,231.289,-61.581,-177.367,6.789,148.482
C02573=1194.956,231.537,-61.607,-177.364,6.791,148.481
C02574=1194.952,231.786,-61.633,-177.362,6.793,148.481
C02575=1194.948,232.035,-61.659,-177.359,6.795,148.481
C02576=1194.943,232.283,-61.684,-177.357,6.798,148.481
C02577=1194.939,232.532,-61.710,-177.354,6.800,148.481
C02578=1194.935,232.781,-61.735,-177.351,6.802,148.480
C02579=1194.929,233.029,-61.761,-177.349,6.804,148.480
C02580=1194.925,233.278,-61.787,-177.346,6.806,148.480
C02581=1194.921,233.527,-61.813,-177.344,6.808,148.480
C02582=1194.916,233.776,-61.839,-177.341,6.810,148.479
C02583=1194.912,234.024,-61.864,-177.338,6.813,148.479
C02584=1194.907,234.272,-61.890,-177.336,6.815,148.479
C02585=1194.902,234.522,-61.916,-177.333,6.817,148.479
C02586=1194.898,234.770,-61.942,-177.331,6.820,148.479
C02587=1194.894,235.018,-61.968,-177.328,6.822,148.478
C02588=1194.889,235.267,-61.994,-177.325,6.824,148.478
C02589=1194.885,235.515,-62.020,-177.323,6.826,148.478
C02590=1194.881,235.764,-62.045,-177.320,6.828,148.478
C02591=1194.875,236.013,-62.071,-177.318,6.831,148.477
C02592=1194.871,236.262,-62.097,-177.315,6.832,148.477
C02593=1194.867,236.533,-62.126,-177.312,6.835,148.477
C02594=1194.862,236.804,-62.153,-177.310,6.837,148.477
C02595=1194.856,237.076,-62.183,-177.307,6.840,148.476
C02596=1194.852,237.347,-62.211,-177.303,6.843,148.476
C02597=1194.847,237.596,-62.237,-177.301,6.845,148.476
C02598=1194.843,237.845,-62.262,-177.299,6.847,148.476
C02599=1194.838,238.093,-62.289,-177.296,6.850,148.476
C02600=1194.834,238.342,-62.315,-177.293,6.851,148.475
C02601=1194.830,238.591,-62.341,-177.291,6.854,148.475
C02602=1194.826,238.839,-62.367,-177.288,6.856,148.475
C02603=1194.821,239.088,-62.393,-177.285,6.858,148.475
C02604=1194.816,239.336,-62.419,-177.283,6.860,148.475
C02605=1194.812,239.584,-62.445,-177.280,6.863,148.474
C02606=1194.807,239.833,-62.472,-177.278,6.865,148.474
C02607=1194.803,240.082,-62.497,-177.275,6.867,148.474
C02608=1194.799,240.330,-62.524,-177.273,6.869,148.474
C02609=1194.794,240.579,-62.550,-177.270,6.872,148.473
C02610=1194.790,240.828,-62.576,-177.268,6.874,148.473
C02611=1194.784,241.076,-62.603,-177.265,6.876,148.473
C02612=1194.780,241.325,-62.628,-177.262,6.879,148.473
C02613=1194.776,241.573,-62.655,-177.260,6.880,148.473
C02614=1194.771,241.822,-62.681,-177.257,6.883,148.473
C02615=1194.767,242.071,-62.707,-177.254,6.885,148.472
C02616=1194.762,242.319,-62.734,-177.252,6.887,148.472
C02617=1194.758,242.568,-62.760,-177.249,6.889,148.472
C02618=1194.754,242.816,-62.786,-177.246,6.892,148.472
C02619=1194.749,243.065,-62.813,-177.244,6.894,148.472
C02620=1194.745,243.313,-62.839,-177.241,6.896,148.471
C02621=1194.740,243.562,-62.865,-177.239,6.899,148.471
C02622=1194.736,243.810,-62.891,-177.236,6.901,148.471
C02623=1194.731,244.059,-62.918,-177.233,6.904,148.471
C02624=1194.727,244.308,-62.944,-177.231,6.906,148.470
C02625=1194.722,244.556,-62.971,-177.228,6.908,148.470
C02626=1194.718,244.805,-62.997,-177.225,6.910,148.470
C02627=1194.713,245.053,-63.024,-177.223,6.913,148.470
C02628=1194.709,245.302,-63.050,-177.221,6.914,148.470
C02629=1194.705,245.551,-63.077,-177.218,6.917,148.470
C02630=1194.701,245.799,-63.103,-177.216,6.920,148.469
C02631=1194.696,246.048,-63.130,-177.213,6.921,148.469
C02632=1194.692,246.296,-63.156,-177.210,6.924,148.469
C02633=1194.687,246.545,-63.183,-177.208,6.926,148.469
C02634=1194.683,246.793,-63.209,-177.205,6.928,148.469
C02635=1194.678,247.042,-63.236,-177.202,6.931,148.468
C02636=1194.674,247.291,-63.262,-177.200,6.933,148.468
C02637=1194.669,247.539,-63.289,-177.197,6.936,148.468
C02638=1194.665,247.788,-63.316,-177.195,6.938,148.468
C02639=1194.661,248.036,-63.342,-177.192,6.940,148.468
C02640=1194.656,248.285,-63.369,-177.189,6.943,148.468
C02641=1194.652,248.533,-63.395,-177.187,6.945,148.467
C02642=1194.647,248.782,-63.422,-177.185,6.947,148.467
C02643=1194.643,249.030,-63.449,-177.181,6.950,148.467
C02644=1194.638,249.279,-63.475,-177.179,6.952,148.467
C02645=1194.634,249.527,-63.502,-177.177,6.955,148.467
C02646=1194.629,249.776,-63.529,-177.174,6.957,148.466
C02647=1194.625,250.024,-63.556,-177.172,6.959,148.466
C02648=1194.620,250.273,-63.583,-177.169,6.961,148.466
C02649=1194.616,250.521,-63.610,-177.166,6.964,148.466
C02650=1194.612,250.770,-63.636,-177.163,6.966,148.466
C02651=1194.607,251.018,-63.663,-177.161,6.968,148.466
C02652=1194.602,251.267,-63.690,-177.158,6.970,148.465
C02653=1194.598,251.515,-63.716,-177.156,6.973,148.465
C02654=1194.594,251.764,-63.743,-177.154,6.975,148.465
C02655=1194.589,252.012,-63.770,-177.150,6.978,148.465
C02656=1194.584,252.261,-63.797,-177.148,6.980,148.465
C02657=1194.581,252.509,-63.824,-177.146,6.982,148.464
C02658=1194.576,252.758,-63.851,-177.143,6.985,148.464
C02659=1194.572,253.006,-63.878,-177.141,6.987,148.464
C02660=1194.567,253.255,-63.905,-177.137,6.990,148.464
C02661=1194.563,253.503,-63.932,-177.135,6.992,148.464
C02662=1194.559,253.752,-63.959,-177.133,6.994,148.464
C02663=1194.554,254.000,-63.986,-177.130,6.997,148.464
C02664=1194.549,254.249,-64.013,-177.127,6.999,148.463
C02665=1194.545,254.497,-64.039,-177.125,7.002,148.463
C02666=1194.541,254.746,-64.067,-177.122,7.004,148.463
C02667=1194.537,254.995,-64.094,-177.119,7.007,148.463
C02668=1194.532,255.243,-64.121,-177.117,7.009,148.463
C02669=1194.527,255.492,-64.148,-177.115,7.011,148.463
C02670=1194.523,255.740,-64.175,-177.112,7.014,148.462
C02671=1194.519,255.988,-64.202,-177.110,7.016,148.462
C02672=1194.514,256.237,-64.229,-177.106,7.018,148.462
C02673=1194.510,256.485,-64.257,-177.104,7.021,148.462
C02674=1194.506,256.734,-64.284,-177.102,7.024,148.462
C02675=1194.501,256.982,-64.311,-177.099,7.025,148.462
C02676=1194.496,257.231,-64.338,-177.096,7.028,148.462
C02677=1194.492,257.479,-64.365,-177.094,7.030,148.461
C02678=1194.488,257.728,-64.392,-177.091,7.032,148.461
C02679=1194.483,257.976,-64.420,-177.089,7.035,148.461
C02680=1194.479,258.224,-64.447,-177.086,7.037,148.461
C02681=1194.475,258.473,-64.474,-177.083,7.040,148.461
C02682=1194.470,258.721,-64.501,-177.081,7.042,148.461
C02683=1194.466,258.970,-64.529,-177.078,7.045,148.460
C02684=1194.462,259.219,-64.556,-177.076,7.047,148.460
C02685=1194.457,259.467,-64.583,-177.073,7.050,148.460
C02686=1194.452,259.716,-64.610,-177.071,7.052,148.460
C02687=1194.448,259.963,-64.638,-177.068,7.054,148.460
C02688=1194.444,260.213,-64.665,-177.066,7.057,148.460
C02689=1194.439,260.461,-64.692,-177.063,7.059,148.460
C02690=1194.435,260.709,-64.720,-177.060,7.062,148.459
C02691=1194.430,260.957,-64.747,-177.058,7.064,148.459
C02692=1194.426,261.207,-64.775,-177.055,7.067,148.459
C02693=1194.422,261.455,-64.802,-177.053,7.069,148.459
C02694=1194.417,261.703,-64.830,-177.050,7.072,148.459
C02695=1194.413,261.951,-64.857,-177.047,7.074,148.459
C02696=1194.409,262.200,-64.885,-177.045,7.077,148.459
C02697=1194.404,262.473,-64.915,-177.042,7.080,148.458
C02698=1194.399,262.746,-64.946,-177.039,7.082,148.458
C02699=1194.394,263.018,-64.975,-177.036,7.085,148.458
C02700=1194.389,263.291,-65.006,-177.033,7.088,148.458
C02701=1194.385,263.540,-65.033,-177.031,7.091,148.458
C02702=1194.381,263.788,-65.061,-177.028,7.092,148.458
C02703=1194.376,264.037,-65.088,-177.026,7.095,148.458
C02704=1194.372,264.285,-65.116,-177.023,7.098,148.458
C02705=1194.367,264.534,-65.144,-177.021,7.099,148.457
C02706=1194.362,264.782,-65.172,-177.018,7.102,148.457
C02707=1194.358,265.031,-65.199,-177.016,7.105,148.457
C02708=1194.354,265.279,-65.227,-177.013,7.108,148.457
C02709=1194.350,265.527,-65.255,-177.010,7.109,148.457
C02710=1194.346,265.776,-65.282,-177.008,7.112,148.457
C02711=1194.341,266.024,-65.310,-177.006,7.115,148.457
C02712=1194.336,266.273,-65.337,-177.002,7.117,148.456
C02713=1194.332,266.521,-65.366,-177.000,7.119,148.456
C02714=1194.328,266.769,-65.393,-176.998,7.122,148.456
C02715=1194.323,267.018,-65.420,-176.995,7.125,148.456
C02716=1194.319,267.266,-65.449,-176.992,7.127,148.456
C02717=1194.314,267.514,-65.477,-176.989,7.130,148.456
C02718=1194.310,267.763,-65.504,-176.987,7.132,148.456
C02719=1194.306,268.011,-65.532,-176.984,7.135,148.455
C02720=1194.302,268.259,-65.560,-176.982,7.137,148.455
C02721=1194.297,268.509,-65.588,-176.979,7.140,148.455
C02722=1194.292,268.757,-65.616,-176.977,7.142,148.455
C02723=1194.288,269.005,-65.644,-176.974,7.145,148.455
C02724=1194.284,269.253,-65.672,-176.972,7.147,148.455
C02725=1194.279,269.502,-65.699,-176.969,7.150,148.455
C02726=1194.275,269.751,-65.727,-176.967,7.152,148.455
C02727=1194.271,269.998,-65.755,-176.964,7.155,148.455
C02728=1194.266,270.247,-65.784,-176.962,7.157,148.454
C02729=1194.262,270.495,-65.812,-176.959,7.160,148.454
C02730=1194.257,270.744,-65.839,-176.957,7.162,148.454
C02731=1194.253,270.993,-65.868,-176.954,7.165,148.454
C02732=1194.249,271.240,-65.895,-176.951,7.167,148.454
C02733=1194.245,271.489,-65.923,-176.949,7.170,148.454
C02734=1194.240,271.737,-65.952,-176.946,7.173,148.454
C02735=1194.236,271.986,-65.980,-176.943,7.175,148.454
C02736=1194.232,272.234,-66.008,-176.941,7.178,148.454
C02737=1194.227,272.483,-66.036,-176.938,7.180,148.454
C02738=1194.223,272.730,-66.064,-176.936,7.183,148.453
C02739=1194.219,272.979,-66.092,-176.933,7.185,148.453
C02740=1194.214,273.227,-66.121,-176.930,7.188,148.453
C02741=1194.210,273.476,-66.148,-176.928,7.190,148.453
C02742=1194.205,273.725,-66.177,-176.926,7.193,148.453
C02743=1194.201,273.973,-66.205,-176.923,7.196,148.453
C02744=1194.196,274.221,-66.233,-176.920,7.198,148.453
C02745=1194.192,274.469,-66.262,-176.918,7.201,148.453
C02746=1194.188,274.717,-66.290,-176.915,7.203,148.453
C02747=1194.184,274.966,-66.318,-176.913,7.206,148.453
C02748=1194.179,275.214,-66.346,-176.910,7.209,148.452
C02749=1194.175,275.463,-66.375,-176.907,7.211,148.452
C02750=1194.170,275.711,-66.403,-176.905,7.213,148.452
C02751=1194.166,275.960,-66.432,-176.902,7.216,148.452
C02752=1194.162,276.207,-66.459,-176.900,7.219,148.452
C02753=1194.157,276.456,-66.488,-176.898,7.222,148.452
C02754=1194.153,276.705,-66.516,-176.894,7.224,148.452
C02755=1194.148,276.953,-66.545,-176.892,7.226,148.452
C02756=1194.145,277.201,-66.573,-176.890,7.229,148.452
C02757=1194.140,277.449,-66.602,-176.887,7.232,148.452
C02758=1194.136,277.698,-66.630,-176.885,7.235,148.451
C02759=1194.131,277.946,-66.658,-176.882,7.238,148.451
C02760=1194.126,278.195,-66.687,-176.879,7.240,148.451
C02761=1194.123,278.443,-66.716,-176.877,7.243,148.451
C02762=1194.118,278.691,-66.744,-176.874,7.245,148.451
C02763=1194.114,278.940,-66.772,-176.872,7.248,148.451
C02764=1194.110,279.189,-66.801,-176.869,7.251,148.451
C02765=1194.106,279.436,-66.830,-176.867,7.253,148.451
C02766=1194.101,279.685,-66.858,-176.864,7.256,148.451
C02767=1194.096,279.933,-66.887,-176.862,7.258,148.451
C02768=1194.092,280.181,-66.915,-176.859,7.261,148.451
C02769=1194.088,280.430,-66.944,-176.856,7.264,148.451
C02770=1194.083,280.678,-66.973,-176.854,7.266,148.450
C02771=1194.079,280.926,-67.001,-176.851,7.269,148.450
C02772=1194.075,281.175,-67.030,-176.849,7.271,148.450
C02773=1194.071,281.423,-67.058,-176.846,7.274,148.450
C02774=1194.067,281.671,-67.088,-176.843,7.277,148.450
C02775=1194.062,281.920,-67.116,-176.841,7.279,148.450
C02776=1194.057,282.168,-67.145,-176.838,7.282,148.450
C02777=1194.054,282.416,-67.173,-176.836,7.284,148.450
C02778=1194.049,282.665,-67.202,-176.834,7.287,148.450
C02779=1194.044,282.912,-67.231,-176.831,7.290,148.450
C02780=1194.041,283.161,-67.259,-176.828,7.292,148.450
C02781=1194.036,283.409,-67.289,-176.826,7.295,148.449
C02782=1194.031,283.657,-67.317,-176.823,7.298,148.449
C02783=1194.027,283.906,-67.346,-176.821,7.300,148.449
C02784=1194.023,284.154,-67.375,-176.818,7.303,148.449
C02785=1194.019,284.402,-67.404,-176.816,7.305,148.449
C02786=1194.014,284.651,-67.433,-176.813,7.308,148.449
C02787=1194.010,284.899,-67.462,-176.810,7.311,148.449
C02788=1194.005,285.148,-67.491,-176.808,7.314,148.449
C02789=1194.001,285.395,-67.519,-176.805,7.316,148.449
C02790=1193.997,285.644,-67.548,-176.802,7.319,148.449
C02791=1193.993,285.892,-67.578,-176.800,7.321,148.449
C02792=1193.988,286.141,-67.606,-176.798,7.324,148.449
C02793=1193.983,286.389,-67.635,-176.795,7.327,148.449
C02794=1193.980,286.637,-67.664,-176.793,7.330,148.449
C02795=1193.975,286.886,-67.693,-176.790,7.333,148.449
C02796=1193.971,287.134,-67.722,-176.788,7.335,148.449
C02797=1193.966,287.381,-67.752,-176.785,7.338,148.449
C02798=1193.962,287.630,-67.780,-176.782,7.341,148.448
C02799=1193.958,287.879,-67.810,-176.780,7.343,148.448
C02800=1193.954,288.127,-67.839,-176.778,7.346,148.448
C02801=1193.949,288.401,-67.871,-176.774,7.349,148.448
C02802=1193.944,288.676,-67.902,-176.772,7.352,148.448
C02803=1193.939,288.950,-67.936,-176.769,7.355,148.448
C02804=1193.935,289.225,-67.967,-176.766,7.358,148.448
C02805=1193.930,289.473,-67.997,-176.764,7.361,148.448
C02806=1193.926,289.721,-68.026,-176.761,7.363,148.448
C02807=1193.921,289.969,-68.055,-176.759,7.366,148.448
C02808=1193.917,290.218,-68.084,-176.756,7.369,148.448
C02809=1193.913,290.466,-68.114,-176.754,7.371,148.448
C02810=1193.909,290.714,-68.143,-176.751,7.374,148.448
C02811=1193.904,290.962,-68.173,-176.748,7.377,148.448
C02812=1193.900,291.211,-68.202,-176.746,7.379,148.448
C02813=1193.895,291.458,-68.231,-176.743,7.382,148.447
C02814=1193.891,291.707,-68.260,-176.740,7.385,148.447
C02815=1193.887,291.955,-68.289,-176.738,7.387,148.447
C02816=1193.883,292.204,-68.319,-176.736,7.390,148.447
C02817=1193.878,292.452,-68.348,-176.733,7.393,148.447
C02818=1193.874,292.700,-68.378,-176.731,7.395,148.447
C02819=1193.870,292.948,-68.407,-176.728,7.398,148.447
C02820=1193.866,293.197,-68.437,-176.725,7.401,148.447
C02821=1193.861,293.444,-68.466,-176.723,7.404,148.447
C02822=1193.857,293.693,-68.495,-176.720,7.407,148.447
C02823=1193.853,293.941,-68.525,-176.718,7.410,148.447
C02824=1193.849,294.189,-68.554,-176.716,7.412,148.447
C02825=1193.844,294.437,-68.583,-176.713,7.415,148.447
C02826=1193.840,294.686,-68.613,-176.710,7.418,148.447
C02827=1193.836,294.934,-68.642,-176.707,7.421,148.447
C02828=1193.831,295.182,-68.672,-176.705,7.423,148.447
C02829=1193.827,295.431,-68.702,-176.703,7.426,148.447
C02830=1193.823,295.679,-68.731,-176.700,7.429,148.447
C02831=1193.819,295.927,-68.761,-176.698,7.431,148.447
C02832=1193.815,296.175,-68.791,-176.695,7.434,148.447
C02833=1193.810,296.423,-68.820,-176.692,7.437,148.447
C02834=1193.806,296.671,-68.850,-176.690,7.439,148.447
C02835=1193.801,296.920,-68.880,-176.687,7.442,148.447
C02836=1193.797,297.168,-68.909,-176.685,7.445,148.447
C02837=1193.792,297.416,-68.938,-176.683,7.448,148.447
C02838=1193.789,297.664,-68.969,-176.680,7.451,148.447
C02839=1193.784,297.912,-68.998,-176.678,7.454,148.447
C02840=1193.780,298.160,-69.027,-176.675,7.457,148.447
C02841=1193.775,298.409,-69.058,-176.673,7.459,148.447
C02842=1193.771,298.657,-69.087,-176.670,7.462,148.447
C02843=1193.767,298.905,-69.117,-176.667,7.465,148.447
C02844=1193.763,299.153,-69.147,-176.665,7.467,148.447
C02845=1193.758,299.401,-69.177,-176.663,7.470,148.447
C02846=1193.754,299.649,-69.207,-176.660,7.473,148.447
C02847=1193.750,299.897,-69.236,-176.657,7.476,148.447
C02848=1193.745,300.146,-69.266,-176.655,7.478,148.446
C02849=1193.742,300.395,-69.296,-176.652,7.481,148.446
C02850=1193.738,300.643,-69.326,-176.650,7.484,148.446
C02851=1193.733,300.891,-69.356,-176.647,7.487,148.446
C02852=1193.729,301.139,-69.387,-176.645,7.490,148.446
C02853=1193.725,301.387,-69.416,-176.642,7.493,148.446
C02854=1193.721,301.635,-69.445,-176.640,7.496,148.446
C02855=1193.716,301.883,-69.476,-176.638,7.498,148.446
C02856=1193.712,302.131,-69.506,-176.635,7.501,148.446
C02857=1193.708,302.379,-69.536,-176.632,7.504,148.446
C02858=1193.703,302.628,-69.566,-176.630,7.506,148.446
C02859=1193.699,302.876,-69.595,-176.627,7.509,148.446
C02860=1193.694,303.124,-69.626,-176.625,7.512,148.446
C02861=1193.690,303.372,-69.656,-176.622,7.515,148.446
C02862=1193.686,303.620,-69.686,-176.620,7.518,148.446
C02863=1193.681,303.868,-69.716,-176.618,7.521,148.446
C02864=1193.677,304.116,-69.746,-176.615,7.524,148.446
C02865=1193.673,304.365,-69.776,-176.613,7.526,148.446
C02866=1193.669,304.613,-69.807,-176.610,7.529,148.446
C02867=1193.665,304.861,-69.837,-176.607,7.532,148.446
C02868=1193.660,305.109,-69.867,-176.605,7.535,148.446
C02869=1193.656,305.357,-69.897,-176.603,7.537,148.446
C02870=1193.651,305.605,-69.927,-176.600,7.540,148.446
C02871=1193.648,305.853,-69.957,-176.598,7.544,148.446
C02872=1193.643,306.102,-69.987,-176.595,7.547,148.446
C02873=1193.639,306.350,-70.018,-176.593,7.549,148.446
C02874=1193.635,306.598,-70.048,-176.590,7.552,148.446
C02875=1193.631,306.846,-70.078,-176.587,7.555,148.446
C02876=1193.626,307.094,-70.109,-176.585,7.558,148.446
C02877=1193.622,307.342,-70.139,-176.583,7.560,148.446
C02878=1193.617,307.590,-70.169,-176.580,7.563,148.446
C02879=1193.614,307.839,-70.199,-176.578,7.566,148.446
C02880=1193.609,308.087,-70.230,-176.575,7.569,148.446
C02881=1193.605,308.334,-70.260,-176.573,7.572,148.446
C02882=1193.601,308.583,-70.290,-176.570,7.575,148.446
C02883=1193.596,308.831,-70.321,-176.568,7.578,148.447
C02884=1193.592,309.079,-70.351,-176.565,7.581,148.447
C02885=1193.588,309.327,-70.382,-176.563,7.583,148.446
C02886=1193.584,309.576,-70.412,-176.560,7.586,148.446
C02887=1193.579,309.823,-70.443,-176.558,7.589,148.446
C02888=1193.575,310.071,-70.473,-176.555,7.592,148.447
C02889=1193.571,310.320,-70.504,-176.553,7.595,148.447
C02890=1193.567,310.568,-70.535,-176.550,7.598,148.447
C02891=1193.563,310.815,-70.565,-176.548,7.601,148.447
C02892=1193.558,311.064,-70.595,-176.546,7.604,148.447
C02893=1193.553,311.312,-70.626,-176.543,7.606,148.447
C02894=1193.550,311.560,-70.656,-176.541,7.609,148.447
C02895=1193.545,311.808,-70.687,-176.538,7.612,148.447
C02896=1193.541,312.056,-70.718,-176.535,7.615,148.447
C02897=1193.537,312.304,-70.748,-176.534,7.618,148.447
C02898=1193.533,312.552,-70.779,-176.531,7.621,148.447
C02899=1193.528,312.800,-70.810,-176.528,7.624,148.447
C02900=1193.524,313.048,-70.841,-176.525,7.627,148.447
C02901=1193.520,313.297,-70.871,-176.524,7.629,148.447
C02902=1193.516,313.545,-70.902,-176.521,7.632,148.447
C02903=1193.511,313.793,-70.933,-176.518,7.635,148.447
C02904=1193.507,314.040,-70.963,-176.516,7.638,148.447
C02905=1193.502,314.317,-70.998,-176.513,7.642,148.447
C02906=1193.497,314.594,-71.032,-176.511,7.645,148.447
C02907=1193.493,314.870,-71.066,-176.508,7.648,148.447
C02908=1193.488,315.146,-71.101,-176.505,7.652,148.447
C02909=1193.484,315.394,-71.132,-176.503,7.654,148.447
C02910=1193.480,315.642,-71.162,-176.500,7.657,148.447
C02911=1193.476,315.890,-71.193,-176.498,7.660,148.447
C02912=1193.472,316.139,-71.224,-176.495,7.663,148.447
C02913=1193.467,316.387,-71.255,-176.493,7.666,148.447
C02914=1193.463,316.635,-71.285,-176.491,7.669,148.447
C02915=1193.459,316.883,-71.316,-176.488,7.672,148.447
C02916=1193.455,317.130,-71.347,-176.486,7.675,148.448
C02917=1193.451,317.379,-71.378,-176.483,7.678,148.448
C02918=1193.446,317.627,-71.409,-176.481,7.680,148.448
C02919=1193.442,317.875,-71.440,-176.479,7.683,148.448
C02920=1193.438,318.123,-71.472,-176.476,7.686,148.448
C02921=1193.433,318.371,-71.503,-176.473,7.689,148.448
C02922=1193.429,318.619,-71.533,-176.472,7.692,148.448
C02923=1193.426,318.867,-71.564,-176.469,7.695,148.448
C02924=1193.421,319.115,-71.595,-176.466,7.698,148.448
C02925=1193.417,319.363,-71.626,-176.464,7.701,148.448
C02926=1193.413,319.611,-71.657,-176.461,7.704,148.448
C02927=1193.408,319.859,-71.689,-176.460,7.707,148.448
C02928=1193.404,320.107,-71.720,-176.457,7.710,148.448
C02929=1193.400,320.355,-71.751,-176.454,7.713,148.448
C02930=1193.396,320.603,-71.782,-176.452,7.716,148.448
C02931=1193.391,320.851,-71.813,-176.449,7.719,148.448
C02932=1193.387,321.100,-71.844,-176.447,7.721,148.448
C02933=1193.383,321.347,-71.876,-176.445,7.725,148.449
C02934=1193.379,321.596,-71.907,-176.442,7.728,148.449
C02935=1193.375,321.843,-71.938,-176.440,7.731,148.449
C02936=1193.370,322.091,-71.969,-176.437,7.734,148.449
C02937=1193.366,322.340,-72.000,-176.435,7.736,148.449
C02938=1193.362,322.587,-72.032,-176.433,7.740,148.449
C02939=1193.358,322.836,-72.063,-176.430,7.743,148.449
C02940=1193.354,323.083,-72.094,-176.428,7.746,148.449
C02941=1193.350,323.332,-72.126,-176.425,7.749,148.449
C02942=1193.345,323.579,-72.157,-176.424,7.751,148.449
C02943=1193.341,323.828,-72.188,-176.421,7.754,148.449
C02944=1193.337,324.075,-72.220,-176.418,7.757,148.449
C02945=1193.333,324.323,-72.251,-176.416,7.761,148.450
C02946=1193.329,324.571,-72.282,-176.413,7.764,148.450
C02947=1193.325,324.819,-72.314,-176.412,7.766,148.450
C02948=1193.320,325.067,-72.345,-176.409,7.769,148.450
C02949=1193.317,325.315,-72.377,-176.407,7.773,148.450
C02950=1193.312,325.562,-72.408,-176.404,7.776,148.450
C02951=1193.307,325.811,-72.440,-176.402,7.779,148.450
C02952=1193.304,326.059,-72.472,-176.399,7.781,148.450
C02953=1193.299,326.307,-72.503,-176.397,7.785,148.450
C02954=1193.295,326.555,-72.534,-176.395,7.788,148.450
C02955=1193.291,326.803,-72.566,-176.392,7.791,148.450
C02956=1193.287,327.051,-72.597,-176.390,7.794,148.450
C02957=1193.283,327.299,-72.628,-176.388,7.796,148.451
C02958=1193.278,327.547,-72.661,-176.385,7.799,148.451
C02959=1193.274,327.794,-72.692,-176.383,7.803,148.451
C02960=1193.270,328.043,-72.724,-176.380,7.806,148.451
C02961=1193.266,328.291,-72.755,-176.378,7.809,148.451
C02962=1193.262,328.539,-72.787,-176.376,7.811,148.451
C02963=1193.258,328.787,-72.819,-176.374,7.815,148.451
C02964=1193.253,329.035,-72.850,-176.371,7.818,148.451
C02965=1193.249,329.283,-72.882,-176.369,7.821,148.451
C02966=1193.246,329.531,-72.914,-176.367,7.824,148.452
C02967=1193.241,329.779,-72.946,-176.364,7.826,148.452
C02968=1193.237,330.027,-72.978,-176.362,7.830,148.452
C02969=1193.233,330.274,-73.009,-176.359,7.833,148.452
C02970=1193.229,330.523,-73.040,-176.357,7.836,148.452
C02971=1193.224,330.771,-73.073,-176.355,7.839,148.452
C02972=1193.220,331.018,-73.104,-176.353,7.842,148.452
C02973=1193.216,331.266,-73.136,-176.351,7.845,148.452
C02974=1193.212,331.514,-73.168,-176.348,7.848,148.452
C02975=1193.207,331.762,-73.200,-176.346,7.851,148.453
C02976=1193.204,332.010,-73.232,-176.343,7.855,148.453
C02977=1193.199,332.257,-73.263,-176.341,7.858,148.453
C02978=1193.195,332.506,-73.296,-176.339,7.860,148.453
C02979=1193.191,332.754,-73.328,-176.337,7.863,148.453
C02980=1193.187,333.001,-73.359,-176.334,7.866,148.453
C02981=1193.182,333.249,-73.391,-176.332,7.870,148.453
C02982=1193.179,333.497,-73.423,-176.329,7.873,148.453
C02983=1193.174,333.745,-73.455,-176.328,7.875,148.454
C02984=1193.170,333.993,-73.487,-176.325,7.879,148.454
C02985=1193.166,334.241,-73.519,-176.323,7.882,148.454
C02986=1193.162,334.490,-73.552,-176.320,7.885,148.454
C02987=1193.157,334.737,-73.583,-176.318,7.888,148.454
C02988=1193.153,334.985,-73.615,-176.316,7.892,148.454
C02989=1193.149,335.233,-73.647,-176.314,7.894,148.454
C02990=1193.145,335.481,-73.679,-176.311,7.897,148.455
C02991=1193.141,335.728,-73.712,-176.309,7.901,148.455
C02992=1193.137,335.976,-73.744,-176.307,7.904,148.455
C02993=1193.133,336.225,-73.776,-176.304,7.907,148.455
C02994=1193.128,336.472,-73.808,-176.303,7.909,148.455
C02995=1193.124,336.720,-73.840,-176.300,7.913,148.455
C02996=1193.120,336.968,-73.872,-176.298,7.916,148.455
C02997=1193.116,337.216,-73.905,-176.295,7.919,148.456
C02998=1193.112,337.464,-73.937,-176.293,7.922,148.456
C02999=1193.107,337.712,-73.969,-176.291,7.926,148.456
C03000=1193.104,337.960,-74.001,-176.289,7.928,148.456
C03001=1193.100,338.208,-74.034,-176.287,7.931,148.456
C03002=1193.095,338.455,-74.066,-176.284,7.935,148.457
C03003=1193.091,338.703,-74.098,-176.282,7.938,148.457
C03004=1193.087,338.951,-74.130,-176.279,7.941,148.457
C03005=1193.083,339.199,-74.163,-176.278,7.943,148.457
C03006=1193.079,339.447,-74.195,-176.276,7.947,148.457
C03007=1193.074,339.695,-74.227,-176.273,7.950,148.457
C03008=1193.071,339.942,-74.259,-176.271,7.953,148.458
C03009=1193.066,340.221,-74.297,-176.269,7.957,148.458
C03010=1193.061,340.500,-74.332,-176.266,7.960,148.458
C03011=1193.056,340.779,-74.369,-176.263,7.964,148.458
C03012=1193.052,341.057,-74.406,-176.261,7.967,148.458
C03013=1193.048,341.305,-74.437,-176.259,7.971,148.459
C03014=1193.043,341.552,-74.470,-176.257,7.974,148.459
C03015=1193.039,341.801,-74.503,-176.254,7.977,148.459
C03016=1193.036,342.048,-74.535,-176.253,7.980,148.459
C03017=1193.031,342.297,-74.568,-176.250,7.983,148.459
C03018=1193.027,342.544,-74.601,-176.248,7.986,148.459
C03019=1193.023,342.792,-74.632,-176.246,7.989,148.460
C03020=1193.019,343.039,-74.665,-176.243,7.993,148.460
C03021=1193.014,343.288,-74.698,-176.241,7.996,148.460
C03022=1193.011,343.535,-74.730,-176.239,7.999,148.460
C03023=1193.006,343.783,-74.763,-176.237,8.002,148.460
C03024=1193.002,344.031,-74.796,-176.235,8.005,148.461
C03025=1192.998,344.280,-74.829,-176.233,8.008,148.461
C03026=1192.994,344.526,-74.861,-176.230,8.012,148.461
C03027=1192.989,344.775,-74.893,-176.229,8.014,148.461
C03028=1192.985,345.022,-74.926,-176.226,8.018,148.461
C03029=1192.981,345.270,-74.959,-176.224,8.021,148.462
C03030=1192.977,345.518,-74.991,-176.222,8.024,148.462
C03031=1192.973,345.766,-75.024,-176.220,8.028,148.462
C03032=1192.969,346.014,-75.057,-176.218,8.031,148.462
C03033=1192.965,346.262,-75.090,-176.216,8.033,148.463
C03034=1192.961,346.509,-75.123,-176.214,8.037,148.463
C03035=1192.957,346.758,-75.155,-176.211,8.040,148.463
C03036=1192.953,347.005,-75.188,-176.209,8.043,148.463
C03037=1192.948,347.252,-75.221,-176.207,8.047,148.463
C03038=1192.944,347.500,-75.254,-176.205,8.050,148.464
C03039=1192.940,347.748,-75.286,-176.203,8.053,148.464
C03040=1192.936,347.996,-75.319,-176.201,8.056,148.464
C03041=1192.932,348.244,-75.352,-176.198,8.059,148.464
C03042=1192.928,348.491,-75.385,-176.196,8.063,148.464
C03043=1192.923,348.740,-75.418,-176.194,8.066,148.465
C03044=1192.919,348.987,-75.451,-176.193,8.069,148.465
C03045=1192.915,349.235,-75.484,-176.191,8.072,148.465
C03046=1192.911,349.483,-75.517,-176.188,8.075,148.466
C03047=1192.907,349.730,-75.550,-176.186,8.079,148.466
C03048=1192.903,349.979,-75.582,-176.184,8.082,148.466
C03049=1192.899,350.226,-75.616,-176.182,8.085,148.466
C03050=1192.895,350.474,-75.649,-176.180,8.088,148.466
C03051=1192.890,350.722,-75.682,-176.178,8.091,148.467
C03052=1192.886,350.970,-75.715,-176.176,8.095,148.467
C03053=1192.882,351.217,-75.748,-176.174,8.098,148.467
C03054=1192.878,351.465,-75.781,-176.171,8.101,148.467
C03055=1192.874,351.713,-75.814,-176.170,8.104,148.468
C03056=1192.870,351.961,-75.848,-176.167,8.107,148.468
C03057=1192.866,352.208,-75.881,-176.166,8.111,148.468
C03058=1192.862,352.456,-75.914,-176.163,8.114,148.469
C03059=1192.857,352.704,-75.947,-176.161,8.118,148.469
C03060=1192.853,352.951,-75.980,-176.159,8.121,148.469
C03061=1192.849,353.199,-76.013,-176.158,8.124,148.469
C03062=1192.845,353.447,-76.047,-176.155,8.127,148.470
C03063=1192.841,353.695,-76.080,-176.153,8.130,148.470
C03064=1192.837,353.942,-76.113,-176.151,8.134,148.470
C03065=1192.833,354.191,-76.146,-176.149,8.137,148.470
C03066=1192.829,354.439,-76.180,-176.147,8.141,148.471
C03067=1192.825,354.686,-76.213,-176.145,8.143,148.471
C03068=1192.821,354.934,-76.246,-176.144,8.147,148.471
C03069=1192.817,355.182,-76.279,-176.141,8.150,148.472
C03070=1192.812,355.429,-76.312,-176.139,8.153,148.472
C03071=1192.808,355.677,-76.345,-176.137,8.157,148.472
C03072=1192.804,355.925,-76.378,-176.136,8.160,148.472
C03073=1192.800,356.172,-76.412,-176.134,8.163,148.473
C03074=1192.796,356.420,-76.446,-176.132,8.167,148.473
C03075=1192.792,356.667,-76.479,-176.129,8.170,148.473
C03076=1192.789,356.916,-76.512,-176.128,8.173,148.474
C03077=1192.784,357.164,-76.545,-176.125,8.177,148.474
C03078=1192.780,357.411,-76.579,-176.124,8.180,148.474
C03079=1192.776,357.659,-76.613,-176.122,8.183,148.475
C03080=1192.772,357.907,-76.646,-176.120,8.186,148.475
C03081=1192.767,358.154,-76.679,-176.118,8.190,148.475
C03082=1192.763,358.402,-76.712,-176.116,8.193,148.475
C03083=1192.760,358.650,-76.747,-176.114,8.196,148.476
C03084=1192.756,358.898,-76.780,-176.112,8.199,148.476
C03085=1192.752,359.145,-76.813,-176.110,8.203,148.476
C03086=1192.747,359.393,-76.847,-176.108,8.206,148.477
C03087=1192.743,359.640,-76.881,-176.106,8.210,148.477
C03088=1192.739,359.888,-76.914,-176.105,8.213,148.477
C03089=1192.736,360.136,-76.948,-176.103,8.216,148.478
C03090=1192.732,360.384,-76.981,-176.101,8.220,148.478
C03091=1192.727,360.632,-77.015,-176.099,8.223,148.478
C03092=1192.723,360.879,-77.049,-176.098,8.226,148.479
C03093=1192.719,361.127,-77.082,-176.096,8.229,148.479
C03094=1192.715,361.375,-77.115,-176.093,8.233,148.479
C03095=1192.711,361.622,-77.149,-176.092,8.236,148.480
C03096=1192.706,361.870,-77.183,-176.090,8.239,148.480
C03097=1192.703,362.117,-77.217,-176.088,8.243,148.480
C03098=1192.698,362.365,-77.250,-176.086,8.246,148.481
C03099=1192.695,362.613,-77.284,-176.085,8.250,148.481
C03100=1192.690,362.861,-77.318,-176.083,8.252,148.482
C03101=1192.687,363.108,-77.352,-176.081,8.256,148.482
C03102=1192.682,363.356,-77.385,-176.079,8.260,148.482
C03103=1192.678,363.604,-77.420,-176.078,8.262,148.483
C03104=1192.674,363.851,-77.453,-176.076,8.266,148.483
C03105=1192.670,364.099,-77.487,-176.074,8.269,148.483
C03106=1192.666,364.346,-77.520,-176.073,8.272,148.484
C03107=1192.662,364.594,-77.555,-176.071,8.276,148.484
C03108=1192.658,364.842,-77.588,-176.069,8.279,148.484
C03109=1192.654,365.089,-77.622,-176.068,8.282,148.485
C03110=1192.650,365.337,-77.656,-176.066,8.286,148.485
C03111=1192.646,365.585,-77.690,-176.064,8.289,148.486
C03112=1192.642,365.832,-77.724,-176.063,8.292,148.486
C03113=1192.637,366.113,-77.762,-176.061,8.296,148.487
C03114=1192.633,366.395,-77.801,-176.059,8.300,148.487
C03115=1192.628,366.676,-77.840,-176.057,8.304,148.487
C03116=1192.624,366.957,-77.878,-176.055,8.307,148.488
C03117=1192.620,367.205,-77.912,-176.054,8.310,148.488
C03118=1192.616,367.452,-77.945,-176.052,8.314,148.489
C03119=1192.611,367.699,-77.980,-176.050,8.317,148.489
C03120=1192.608,367.947,-78.014,-176.049,8.320,148.490
C03121=1192.603,368.195,-78.048,-176.047,8.324,148.490
C03122=1192.599,368.442,-78.082,-176.046,8.327,148.490
C03123=1192.595,368.690,-78.117,-176.044,8.330,148.491
C03124=1192.591,368.938,-78.150,-176.043,8.333,148.491
C03125=1192.587,369.185,-78.184,-176.041,8.337,148.492
C03126=1192.583,369.433,-78.218,-176.039,8.340,148.492
C03127=1192.579,369.680,-78.252,-176.038,8.343,148.492
C03128=1192.575,369.928,-78.286,-176.036,8.347,148.493
C03129=1192.571,370.176,-78.320,-176.035,8.350,148.493
C03130=1192.567,370.424,-78.355,-176.034,8.353,148.494
C03131=1192.563,370.671,-78.389,-176.033,8.356,148.494
C03132=1192.559,370.919,-78.424,-176.031,8.360,148.495
C03133=1192.555,371.166,-78.457,-176.030,8.363,148.495
C03134=1192.550,371.414,-78.491,-176.028,8.366,148.496
C03135=1192.547,371.662,-78.525,-176.026,8.369,148.496
C03136=1192.542,371.909,-78.560,-176.025,8.373,148.497
C03137=1192.539,372.157,-78.594,-176.024,8.376,148.497
C03138=1192.535,372.405,-78.629,-176.023,8.379,148.497
C03139=1192.530,372.652,-78.663,-176.021,8.382,148.498
C03140=1192.527,372.900,-78.697,-176.020,8.385,148.498
C03141=1192.522,373.147,-78.732,-176.018,8.389,148.499
C03142=1192.519,373.395,-78.766,-176.017,8.392,148.499
C03143=1192.514,373.643,-78.800,-176.015,8.395,148.500
C03144=1192.510,373.890,-78.834,-176.014,8.399,148.500
C03145=1192.506,374.138,-78.868,-176.013,8.401,148.501
C03146=1192.502,374.386,-78.903,-176.011,8.405,148.501
C03147=1192.499,374.634,-78.937,-176.011,8.408,148.502
C03148=1192.494,374.881,-78.972,-176.009,8.411,148.502
C03149=1192.490,375.128,-79.005,-176.008,8.415,148.502
C03150=1192.486,375.376,-79.040,-176.007,8.418,148.503
C03151=1192.482,375.624,-79.075,-176.006,8.420,148.503
C03152=1192.478,375.871,-79.109,-176.004,8.424,148.504
C03153=1192.474,376.119,-79.143,-176.003,8.427,148.504
C03154=1192.471,376.367,-79.178,-176.002,8.430,148.505
C03155=1192.466,376.614,-79.212,-176.000,8.434,148.506
C03156=1192.462,376.861,-79.247,-176.000,8.437,148.506
C03157=1192.459,377.109,-79.282,-175.998,8.440,148.506
C03158=1192.454,377.356,-79.316,-175.998,8.443,148.507
C03159=1192.450,377.604,-79.351,-175.996,8.446,148.508
C03160=1192.446,377.851,-79.385,-175.995,8.450,148.508
C03161=1192.442,378.099,-79.420,-175.994,8.452,148.508
C03162=1192.438,378.347,-79.454,-175.993,8.455,148.509
C03163=1192.434,378.595,-79.488,-175.991,8.459,148.509
C03164=1192.430,378.842,-79.523,-175.990,8.462,148.510
C03165=1192.426,379.090,-79.558,-175.989,8.465,148.510
C03166=1192.422,379.337,-79.593,-175.988,8.468,148.511
C03167=1192.418,379.584,-79.627,-175.988,8.471,148.512
C03168=1192.414,379.832,-79.661,-175.986,8.474,148.512
C03169=1192.409,380.080,-79.696,-175.985,8.478,148.513
C03170=1192.406,380.327,-79.730,-175.984,8.481,148.513
C03171=1192.402,380.574,-79.765,-175.983,8.484,148.514
C03172=1192.398,380.822,-79.800,-175.982,8.487,148.514
C03173=1192.393,381.070,-79.835,-175.981,8.490,148.515
C03174=1192.390,381.318,-79.869,-175.980,8.493,148.515
C03175=1192.385,381.565,-79.903,-175.979,8.496,148.516
C03176=1192.382,381.813,-79.939,-175.979,8.499,148.516
C03177=1192.377,382.060,-79.973,-175.978,8.502,148.517
C03178=1192.373,382.308,-80.008,-175.977,8.505,148.517
C03179=1192.369,382.555,-80.042,-175.976,8.508,148.518
C03180=1192.366,382.803,-80.078,-175.975,8.511,148.519
C03181=1192.361,383.050,-80.112,-175.974,8.514,148.519
C03182=1192.357,383.298,-80.147,-175.973,8.517,148.519
C03183=1192.354,383.545,-80.182,-175.972,8.520,148.520
C03184=1192.350,383.793,-80.216,-175.971,8.523,148.521
C03185=1192.346,384.041,-80.251,-175.971,8.526,148.521
C03186=1192.341,384.288,-80.286,-175.970,8.529,148.522
C03187=1192.337,384.536,-80.321,-175.969,8.533,148.522
C03188=1192.333,384.783,-80.356,-175.968,8.535,148.523
C03189=1192.330,385.030,-80.391,-175.967,8.538,148.523
C03190=1192.325,385.278,-80.425,-175.966,8.542,148.524
C03191=1192.321,385.526,-80.460,-175.966,8.544,148.525
C03192=1192.317,385.773,-80.495,-175.965,8.547,148.525
C03193=1192.313,386.021,-80.530,-175.964,8.550,148.526
C03194=1192.309,386.269,-80.565,-175.963,8.553,148.526
C03195=1192.306,386.516,-80.599,-175.963,8.556,148.527
C03196=1192.302,386.764,-80.634,-175.962,8.559,148.527
C03197=1192.297,387.010,-80.669,-175.962,8.562,148.528
C03198=1192.294,387.259,-80.704,-175.961,8.565,148.529
C03199=1192.289,387.505,-80.739,-175.960,8.568,148.529
C03200=1192.285,387.754,-80.774,-175.959,8.571,148.530
C03201=1192.281,388.002,-80.809,-175.959,8.573,148.530
C03202=1192.277,388.248,-80.844,-175.958,8.576,148.531
C03203=1192.274,388.496,-80.878,-175.957,8.579,148.531
C03204=1192.270,388.743,-80.914,-175.957,8.582,148.532
C03205=1192.266,388.991,-80.948,-175.956,8.585,148.533
C03206=1192.262,389.239,-80.984,-175.956,8.588,148.533
C03207=1192.257,389.486,-81.018,-175.955,8.590,148.534
C03208=1192.254,389.734,-81.054,-175.955,8.593,148.534
C03209=1192.249,389.981,-81.088,-175.954,8.596,148.535
C03210=1192.245,390.228,-81.124,-175.954,8.599,148.535
C03211=1192.241,390.477,-81.159,-175.953,8.602,148.536
C03212=1192.237,390.723,-81.194,-175.952,8.604,148.536
C03213=1192.233,390.972,-81.229,-175.952,8.607,148.537
C03214=1192.229,391.218,-81.264,-175.951,8.610,148.538
C03215=1192.226,391.466,-81.298,-175.951,8.612,148.538
C03216=1192.222,391.714,-81.334,-175.950,8.615,148.539
C03217=1192.217,391.997,-81.374,-175.950,8.618,148.540
C03218=1192.212,392.280,-81.414,-175.949,8.621,148.540
C03219=1192.208,392.564,-81.454,-175.949,8.625,148.541
C03220=1192.203,392.847,-81.494,-175.948,8.628,148.541
C03221=1192.200,393.094,-81.530,-175.948,8.630,148.542
C03222=1192.196,393.342,-81.565,-175.947,8.633,148.543
C03223=1192.191,393.589,-81.600,-175.947,8.635,148.543
C03224=1192.187,393.837,-81.635,-175.946,8.638,148.544
C03225=1192.184,394.085,-81.670,-175.946,8.641,148.544
C03226=1192.180,394.332,-81.705,-175.945,8.644,148.545
C03227=1192.176,394.580,-81.740,-175.945,8.646,148.546
C03228=1192.171,394.826,-81.775,-175.945,8.649,148.546
C03229=1192.167,395.075,-81.810,-175.944,8.652,148.547
C03230=1192.164,395.322,-81.846,-175.944,8.654,148.547
C03231=1192.159,395.569,-81.881,-175.943,8.657,148.548
C03232=1192.155,395.817,-81.916,-175.943,8.660,148.548
C03233=1192.152,396.064,-81.951,-175.943,8.662,148.549
C03234=1192.148,396.311,-81.986,-175.942,8.665,148.550
C03235=1192.144,396.559,-82.021,-175.942,8.667,148.550
C03236=1192.140,396.807,-82.057,-175.942,8.669,148.551
C03237=1192.136,397.054,-82.092,-175.942,8.672,148.551
C03238=1192.132,397.302,-82.127,-175.941,8.675,148.552
C03239=1192.128,397.549,-82.162,-175.941,8.677,148.553
C03240=1192.124,397.796,-82.198,-175.941,8.680,148.553
C03241=1192.119,398.045,-82.233,-175.940,8.682,148.554
C03242=1192.115,398.292,-82.269,-175.940,8.685,148.554
C03243=1192.111,398.539,-82.304,-175.939,8.687,148.555
C03244=1192.107,398.787,-82.339,-175.939,8.690,148.555
C03245=1192.103,399.034,-82.374,-175.939,8.692,148.556
C03246=1192.099,399.281,-82.409,-175.939,8.695,148.557
C03247=1192.096,399.529,-82.445,-175.938,8.698,148.557
C03248=1192.092,399.777,-82.480,-175.938,8.700,148.558
C03249=1192.087,400.024,-82.515,-175.938,8.702,148.558
C03250=1192.084,400.271,-82.550,-175.938,8.704,148.559
C03251=1192.080,400.519,-82.586,-175.937,8.707,148.559
C03252=1192.076,400.767,-82.621,-175.938,8.709,148.560
C03253=1192.072,401.014,-82.656,-175.937,8.712,148.560
C03254=1192.068,401.261,-82.692,-175.937,8.715,148.561
C03255=1192.064,401.509,-82.728,-175.936,8.717,148.562
C03256=1192.059,401.756,-82.762,-175.936,8.719,148.562
C03257=1192.055,402.004,-82.798,-175.936,8.721,148.563
C03258=1192.052,402.251,-82.833,-175.936,8.724,148.563
C03259=1192.048,402.498,-82.868,-175.936,8.726,148.564
C03260=1192.044,402.746,-82.904,-175.936,8.728,148.564
C03261=1192.040,402.994,-82.939,-175.935,8.731,148.565
C03262=1192.036,403.241,-82.974,-175.935,8.733,148.565
C03263=1192.032,403.488,-83.010,-175.935,8.735,148.566
C03264=1192.028,403.736,-83.046,-175.935,8.737,148.566
C03265=1192.024,403.983,-83.081,-175.935,8.740,148.567
C03266=1192.020,404.230,-83.116,-175.934,8.742,148.568
C03267=1192.016,404.478,-83.151,-175.934,8.745,148.568
C03268=1192.012,404.726,-83.187,-175.934,8.747,148.569
C03269=1192.008,404.973,-83.222,-175.934,8.749,148.569
C03270=1192.004,405.220,-83.258,-175.934,8.751,148.570
C03271=1192.000,405.468,-83.293,-175.933,8.754,148.570
C03272=1191.996,405.715,-83.329,-175.933,8.756,148.571
C03273=1191.992,405.964,-83.364,-175.933,8.758,148.572
C03274=1191.988,406.210,-83.399,-175.933,8.761,148.572
C03275=1191.984,406.458,-83.435,-175.933,8.763,148.573
C03276=1191.980,406.705,-83.470,-175.932,8.765,148.573
C03277=1191.977,406.953,-83.506,-175.932,8.768,148.574
C03278=1191.972,407.200,-83.542,-175.932,8.770,148.574
C03279=1191.968,407.447,-83.577,-175.932,8.772,148.575
C03280=1191.964,407.695,-83.613,-175.931,8.774,148.575
C03281=1191.961,407.942,-83.648,-175.931,8.777,148.576
C03282=1191.956,408.190,-83.683,-175.931,8.779,148.576
C03283=1191.953,408.437,-83.718,-175.931,8.781,148.577
C03284=1191.948,408.685,-83.754,-175.932,8.783,148.578
C03285=1191.945,408.933,-83.790,-175.931,8.785,148.578
C03286=1191.940,409.179,-83.825,-175.931,8.787,148.579
C03287=1191.937,409.427,-83.861,-175.931,8.790,148.579
C03288=1191.933,409.674,-83.896,-175.931,8.792,148.580
C03289=1191.929,409.922,-83.932,-175.930,8.794,148.580
C03290=1191.924,410.169,-83.968,-175.930,8.796,148.581
C03291=1191.921,410.417,-84.003,-175.930,8.798,148.581
C03292=1191.917,410.664,-84.039,-175.930,8.800,148.582
C03293=1191.913,410.912,-84.074,-175.930,8.802,148.582
C03294=1191.909,411.158,-84.109,-175.930,8.805,148.583
C03295=1191.905,411.406,-84.146,-175.929,8.807,148.583
C03296=1191.901,411.654,-84.181,-175.929,8.809,148.584
C03297=1191.897,411.901,-84.217,-175.929,8.811,148.584
C03298=1191.893,412.148,-84.252,-175.929,8.813,148.585
C03299=1191.889,412.396,-84.288,-175.929,8.815,148.585
C03300=1191.885,412.643,-84.324,-175.929,8.817,148.586
C03301=1191.881,412.891,-84.359,-175.929,8.819,148.586
C03302=1191.877,413.139,-84.394,-175.929,8.821,148.587
C03303=1191.873,413.386,-84.429,-175.928,8.823,148.587
C03304=1191.869,413.634,-84.465,-175.928,8.826,148.588
C03305=1191.865,413.881,-84.501,-175.928,8.828,148.588
C03306=1191.862,414.128,-84.537,-175.928,8.829,148.589
C03307=1191.857,414.375,-84.572,-175.928,8.832,148.589
C03308=1191.853,414.623,-84.608,-175.928,8.834,148.590
C03309=1191.849,414.870,-84.644,-175.928,8.836,148.590
C03310=1191.846,415.118,-84.679,-175.928,8.838,148.591
C03311=1191.842,415.365,-84.715,-175.928,8.840,148.591
C03312=1191.837,415.612,-84.751,-175.927,8.842,148.592
C03313=1191.831,415.988,-84.805,-175.928,8.845,148.593
C03314=1191.827,416.364,-84.859,-175.927,8.848,148.593
C03315=1191.827,416.740,-84.913,-175.927,8.851,148.594
C03316=1191.830,417.115,-84.965,-175.927,8.854,148.595
C03317=1191.409,417.116,-85.006,-175.930,8.865,148.599
C03318=1191.406,416.738,-84.952,-175.930,8.861,148.598
C03319=1191.406,416.359,-84.898,-175.930,8.859,148.597
C03320=1191.410,415.980,-84.843,-175.931,8.855,148.596
C03321=1191.415,415.602,-84.789,-175.930,8.853,148.596
C03322=1191.420,415.355,-84.753,-175.931,8.851,148.595
C03323=1191.424,415.107,-84.717,-175.931,8.848,148.595
C03324=1191.428,414.860,-84.682,-175.931,8.847,148.594
C03325=1191.431,414.612,-84.646,-175.931,8.845,148.594
C03326=1191.436,414.364,-84.610,-175.931,8.842,148.593
C03327=1191.440,414.118,-84.575,-175.931,8.840,148.592
C03328=1191.444,413.870,-84.540,-175.931,8.839,148.592
C03329=1191.447,413.623,-84.504,-175.931,8.836,148.591
C03330=1191.452,413.375,-84.468,-175.932,8.834,148.591
C03331=1191.455,413.127,-84.432,-175.932,8.832,148.590
C03332=1191.460,412.880,-84.397,-175.932,8.830,148.590
C03333=1191.463,412.633,-84.362,-175.932,8.828,148.589
C03334=1191.468,412.385,-84.325,-175.932,8.826,148.589
C03335=1191.471,412.138,-84.290,-175.932,8.824,148.588
C03336=1191.476,411.891,-84.255,-175.933,8.821,148.588
C03337=1191.479,411.643,-84.219,-175.932,8.820,148.587
C03338=1191.483,411.396,-84.184,-175.932,8.818,148.587
C03339=1191.487,411.148,-84.147,-175.933,8.815,148.586
C03340=1191.491,410.901,-84.112,-175.933,8.813,148.586
C03341=1191.495,410.654,-84.077,-175.933,8.811,148.585
C03342=1191.499,410.406,-84.041,-175.933,8.809,148.585
C03343=1191.503,410.158,-84.006,-175.933,8.807,148.584
C03344=1191.507,409.910,-83.970,-175.933,8.805,148.584
C03345=1191.512,409.663,-83.935,-175.934,8.803,148.583
C03346=1191.515,409.416,-83.899,-175.934,8.800,148.583
C03347=1191.519,409.168,-83.864,-175.934,8.798,148.582
C03348=1191.523,408.921,-83.828,-175.934,8.797,148.582
C03349=1191.528,408.674,-83.793,-175.934,8.794,148.581
C03350=1191.531,408.426,-83.757,-175.934,8.792,148.580
C03351=1191.535,408.179,-83.721,-175.934,8.790,148.580
C03352=1191.539,407.931,-83.686,-175.934,8.787,148.579
C03353=1191.542,407.684,-83.650,-175.935,8.785,148.579
C03354=1191.547,407.437,-83.615,-175.935,8.783,148.578
C03355=1191.551,407.189,-83.579,-175.935,8.780,148.578
C03356=1191.555,406.942,-83.544,-175.935,8.778,148.577
C03357=1191.559,406.694,-83.509,-175.936,8.776,148.577
C03358=1191.563,406.447,-83.474,-175.935,8.774,148.576
C03359=1191.567,406.199,-83.438,-175.935,8.772,148.576
C03360=1191.570,405.952,-83.402,-175.935,8.770,148.575
C03361=1191.575,405.705,-83.367,-175.936,8.767,148.575
C03362=1191.579,405.457,-83.331,-175.936,8.765,148.574
C03363=1191.582,405.210,-83.296,-175.936,8.763,148.574
C03364=1191.586,404.962,-83.260,-175.936,8.761,148.573
C03365=1191.591,404.715,-83.226,-175.937,8.758,148.572
C03366=1191.594,404.467,-83.190,-175.936,8.756,148.572
C03367=1191.598,404.220,-83.154,-175.937,8.754,148.571
C03368=1191.602,403.972,-83.118,-175.937,8.751,148.571
C03369=1191.607,403.725,-83.083,-175.937,8.749,148.570
C03370=1191.610,403.478,-83.048,-175.937,8.747,148.570
C03371=1191.614,403.230,-83.013,-175.938,8.744,148.569
C03372=1191.619,402.983,-82.978,-175.938,8.742,148.569
C03373=1191.622,402.735,-82.942,-175.938,8.740,148.568
C03374=1191.626,402.488,-82.906,-175.938,8.737,148.567
C03375=1191.630,402.240,-82.871,-175.938,8.735,148.567
C03376=1191.635,401.993,-82.836,-175.939,8.732,148.566
C03377=1191.639,401.745,-82.800,-175.939,8.730,148.566
C03378=1191.642,401.498,-82.765,-175.939,8.727,148.565
C03379=1191.646,401.251,-82.730,-175.939,8.725,148.564
C03380=1191.650,401.003,-82.694,-175.939,8.723,148.564
C03381=1191.654,400.755,-82.659,-175.940,8.720,148.563
C03382=1191.658,400.508,-82.624,-175.940,8.718,148.563
C03383=1191.662,400.261,-82.588,-175.940,8.716,148.562
C03384=1191.666,400.013,-82.553,-175.941,8.713,148.562
C03385=1191.670,399.765,-82.518,-175.941,8.710,148.561
C03386=1191.675,399.518,-82.482,-175.941,8.708,148.561
C03387=1191.678,399.271,-82.447,-175.941,8.706,148.560
C03388=1191.682,399.023,-82.411,-175.942,8.703,148.559
C03389=1191.687,398.776,-82.377,-175.942,8.701,148.559
C03390=1191.690,398.528,-82.341,-175.943,8.698,148.558
C03391=1191.694,398.281,-82.306,-175.942,8.695,148.558
C03392=1191.698,398.034,-82.270,-175.943,8.693,148.557
C03393=1191.702,397.786,-82.236,-175.943,8.691,148.557
C03394=1191.706,397.538,-82.200,-175.944,8.688,148.556
C03395=1191.710,397.291,-82.165,-175.944,8.686,148.555
C03396=1191.714,397.043,-82.130,-175.944,8.683,148.555
C03397=1191.718,396.796,-82.095,-175.944,8.681,148.554
C03398=1191.722,396.549,-82.059,-175.945,8.678,148.554
C03399=1191.726,396.301,-82.025,-175.945,8.675,148.553
C03400=1191.730,396.053,-81.989,-175.945,8.673,148.553
C03401=1191.734,395.807,-81.954,-175.946,8.670,148.552
C03402=1191.738,395.558,-81.919,-175.946,8.668,148.551
C03403=1191.741,395.311,-81.883,-175.946,8.665,148.551
C03404=1191.746,395.064,-81.848,-175.947,8.662,148.550
C03405=1191.750,394.816,-81.813,-175.947,8.660,148.550
C03406=1191.753,394.569,-81.778,-175.947,8.657,148.549
C03407=1191.758,394.322,-81.743,-175.948,8.654,148.548
C03408=1191.762,394.074,-81.708,-175.948,8.652,148.548
C03409=1191.765,393.826,-81.672,-175.949,8.649,148.547
C03410=1191.770,393.579,-81.638,-175.949,8.646,148.547
C03411=1191.774,393.331,-81.602,-175.950,8.643,148.546
C03412=1191.777,393.084,-81.567,-175.950,8.641,148.546
C03413=1191.782,392.836,-81.532,-175.950,8.639,148.545
C03414=1191.786,392.553,-81.491,-175.951,8.636,148.544
C03415=1191.791,392.269,-81.451,-175.951,8.632,148.544
C03416=1191.796,391.986,-81.411,-175.952,8.629,148.543
C03417=1191.800,391.703,-81.372,-175.953,8.626,148.542
C03418=1191.804,391.455,-81.336,-175.953,8.624,148.542
C03419=1191.808,391.208,-81.301,-175.954,8.620,148.541
C03420=1191.812,390.960,-81.266,-175.954,8.618,148.541
C03421=1191.815,390.713,-81.230,-175.955,8.615,148.540
C03422=1191.820,390.465,-81.196,-175.955,8.612,148.539
C03423=1191.824,390.218,-81.160,-175.956,8.610,148.539
C03424=1191.828,389.970,-81.126,-175.957,8.607,148.538
C03425=1191.832,389.723,-81.090,-175.957,8.604,148.538
C03426=1191.836,389.475,-81.056,-175.958,8.601,148.537
C03427=1191.840,389.228,-81.020,-175.958,8.598,148.537
C03428=1191.844,388.980,-80.986,-175.959,8.596,148.536
C03429=1191.848,388.733,-80.951,-175.959,8.592,148.535
C03430=1191.852,388.485,-80.916,-175.960,8.589,148.535
C03431=1191.855,388.238,-80.881,-175.960,8.587,148.534
C03432=1191.860,387.990,-80.846,-175.961,8.584,148.534
C03433=1191.864,387.742,-80.811,-175.962,8.581,148.533
C03434=1191.868,387.495,-80.776,-175.962,8.578,148.532
C03435=1191.872,387.247,-80.741,-175.963,8.576,148.532
C03436=1191.876,387.000,-80.706,-175.963,8.572,148.531
C03437=1191.880,386.752,-80.671,-175.964,8.569,148.531
C03438=1191.883,386.505,-80.636,-175.965,8.567,148.530
C03439=1191.888,386.258,-80.602,-175.966,8.564,148.530
C03440=1191.892,386.010,-80.567,-175.966,8.561,148.529
C03441=1191.896,385.763,-80.532,-175.967,8.558,148.529
C03442=1191.900,385.515,-80.497,-175.968,8.555,148.528
C03443=1191.904,385.268,-80.462,-175.969,8.552,148.527
C03444=1191.908,385.020,-80.427,-175.970,8.549,148.527
C03445=1191.911,384.772,-80.393,-175.970,8.546,148.526
C03446=1191.916,384.525,-80.358,-175.971,8.543,148.526
C03447=1191.920,384.277,-80.323,-175.971,8.540,148.525
C03448=1191.924,384.030,-80.288,-175.972,8.537,148.525
C03449=1191.928,383.782,-80.253,-175.974,8.534,148.524
C03450=1191.932,383.535,-80.219,-175.974,8.531,148.524
C03451=1191.936,383.287,-80.184,-175.975,8.528,148.523
C03452=1191.940,383.040,-80.149,-175.976,8.525,148.522
C03453=1191.944,382.792,-80.114,-175.977,8.522,148.522
C03454=1191.949,382.545,-80.080,-175.978,8.519,148.521
C03455=1191.951,382.297,-80.045,-175.979,8.516,148.521
C03456=1191.956,382.050,-80.010,-175.980,8.513,148.520
C03457=1191.960,381.802,-79.975,-175.980,8.510,148.520
C03458=1191.965,381.554,-79.941,-175.981,8.507,148.519
C03459=1191.968,381.307,-79.905,-175.982,8.504,148.519
C03460=1191.972,381.060,-79.871,-175.984,8.500,148.518
C03461=1191.976,380.812,-79.837,-175.984,8.497,148.518
C03462=1191.981,380.564,-79.802,-175.986,8.494,148.517
C03463=1191.985,380.316,-79.767,-175.987,8.491,148.517
C03464=1191.988,380.070,-79.733,-175.987,8.488,148.516
C03465=1191.992,379.821,-79.698,-175.989,8.485,148.516
C03466=1191.997,379.574,-79.663,-175.989,8.482,148.515
C03467=1192.001,379.326,-79.629,-175.990,8.479,148.514
C03468=1192.004,379.079,-79.595,-175.992,8.475,148.514
C03469=1192.008,378.831,-79.559,-175.993,8.472,148.513
C03470=1192.013,378.584,-79.525,-175.994,8.470,148.513
C03471=1192.016,378.336,-79.490,-175.995,8.466,148.512
C03472=1192.020,378.089,-79.456,-175.996,8.463,148.512
C03473=1192.024,377.841,-79.421,-175.997,8.460,148.511
C03474=1192.028,377.593,-79.387,-175.998,8.457,148.511
C03475=1192.032,377.345,-79.352,-175.999,8.454,148.510
C03476=1192.037,377.098,-79.318,-176.000,8.451,148.510
C03477=1192.040,376.850,-79.284,-176.002,8.447,148.509
C03478=1192.044,376.603,-79.249,-176.003,8.444,148.509
C03479=1192.049,376.356,-79.214,-176.004,8.441,148.508
C03480=1192.052,376.108,-79.180,-176.005,8.437,148.508
C03481=1192.057,375.861,-79.145,-176.007,8.434,148.507
C03482=1192.061,375.613,-79.111,-176.008,8.432,148.507
C03483=1192.064,375.365,-79.077,-176.009,8.428,148.506
C03484=1192.068,375.117,-79.042,-176.010,8.425,148.506
C03485=1192.072,374.870,-79.008,-176.011,8.422,148.505
C03486=1192.077,374.623,-78.973,-176.013,8.418,148.505
C03487=1192.081,374.375,-78.939,-176.014,8.415,148.505
C03488=1192.085,374.128,-78.905,-176.015,8.412,148.504
C03489=1192.089,373.879,-78.870,-176.017,8.409,148.504
C03490=1192.092,373.632,-78.836,-176.018,8.406,148.503
C03491=1192.097,373.385,-78.802,-176.019,8.402,148.503
C03492=1192.101,373.137,-78.767,-176.021,8.399,148.502
C03493=1192.105,372.889,-78.734,-176.022,8.396,148.502
C03494=1192.109,372.641,-78.699,-176.023,8.392,148.501
C03495=1192.113,372.394,-78.665,-176.024,8.390,148.501
C03496=1192.117,372.146,-78.630,-176.026,8.386,148.500
C03497=1192.121,371.899,-78.596,-176.027,8.383,148.500
C03498=1192.125,371.651,-78.562,-176.029,8.379,148.499
C03499=1192.129,371.403,-78.527,-176.030,8.376,148.499
C03500=1192.133,371.156,-78.493,-176.032,8.373,148.498
C03501=1192.137,370.909,-78.459,-176.033,8.370,148.498
C03502=1192.141,370.660,-78.425,-176.035,8.366,148.498
C03503=1192.145,370.413,-78.391,-176.036,8.364,148.497
C03504=1192.150,370.166,-78.357,-176.037,8.360,148.497
C03505=1192.153,369.918,-78.322,-176.039,8.357,148.496
C03506=1192.157,369.670,-78.288,-176.041,8.353,148.496
C03507=1192.162,369.423,-78.255,-176.042,8.350,148.495
C03508=1192.165,369.174,-78.220,-176.044,8.347,148.495
C03509=1192.169,368.927,-78.186,-176.045,8.344,148.495
C03510=1192.174,368.680,-78.152,-176.047,8.340,148.494
C03511=1192.177,368.432,-78.118,-176.048,8.337,148.494
C03512=1192.182,368.184,-78.084,-176.050,8.334,148.493
C03513=1192.186,367.937,-78.050,-176.051,8.330,148.493
C03514=1192.190,367.689,-78.015,-176.053,8.327,148.492
C03515=1192.194,367.441,-77.982,-176.054,8.324,148.492
C03516=1192.198,367.194,-77.948,-176.056,8.321,148.492
C03517=1192.202,366.946,-77.913,-176.057,8.317,148.491
C03518=1192.207,366.665,-77.875,-176.059,8.314,148.491
C03519=1192.212,366.384,-77.837,-176.061,8.310,148.490
C03520=1192.216,366.103,-77.798,-176.063,8.307,148.490
C03521=1192.220,365.822,-77.759,-176.065,8.302,148.489
C03522=1192.224,365.574,-77.726,-176.066,8.299,148.489
C03523=1192.229,365.326,-77.692,-176.068,8.296,148.489
C03524=1192.232,365.079,-77.658,-176.070,8.292,148.488
C03525=1192.236,364.831,-77.624,-176.071,8.289,148.488
C03526=1192.240,364.583,-77.590,-176.073,8.286,148.488
C03527=1192.245,364.336,-77.556,-176.075,8.282,148.487
C03528=1192.248,364.088,-77.523,-176.077,8.279,148.487
C03529=1192.253,363.840,-77.489,-176.078,8.276,148.486
C03530=1192.257,363.593,-77.455,-176.080,8.272,148.486
C03531=1192.261,363.345,-77.421,-176.082,8.270,148.486
C03532=1192.265,363.097,-77.387,-176.084,8.266,148.485
C03533=1192.269,362.850,-77.354,-176.085,8.262,148.485
C03534=1192.273,362.602,-77.320,-176.088,8.259,148.485
C03535=1192.277,362.354,-77.286,-176.089,8.256,148.484
C03536=1192.281,362.107,-77.252,-176.091,8.253,148.484
C03537=1192.285,361.859,-77.219,-176.092,8.249,148.483
C03538=1192.289,361.611,-77.185,-176.094,8.247,148.483
C03539=1192.293,361.364,-77.151,-176.096,8.243,148.483
C03540=1192.297,361.116,-77.117,-176.098,8.240,148.482
C03541=1192.302,360.868,-77.084,-176.100,8.236,148.482
C03542=1192.306,360.621,-77.051,-176.102,8.232,148.482
C03543=1192.309,360.373,-77.016,-176.103,8.230,148.481
C03544=1192.313,360.125,-76.983,-176.105,8.226,148.481
C03545=1192.318,359.878,-76.949,-176.107,8.223,148.481
C03546=1192.322,359.630,-76.916,-176.109,8.219,148.480
C03547=1192.326,359.382,-76.882,-176.110,8.216,148.480
C03548=1192.330,359.135,-76.849,-176.113,8.213,148.480
C03549=1192.333,358.887,-76.815,-176.114,8.209,148.479
C03550=1192.338,358.639,-76.781,-176.117,8.206,148.479
C03551=1192.342,358.391,-76.748,-176.119,8.202,148.479
C03552=1192.346,358.144,-76.714,-176.120,8.200,148.478
C03553=1192.350,357.896,-76.681,-176.122,8.196,148.478
C03554=1192.354,357.648,-76.648,-176.124,8.193,148.478
C03555=1192.358,357.400,-76.614,-176.126,8.190,148.478
C03556=1192.362,357.153,-76.581,-176.128,8.186,148.477
C03557=1192.367,356.905,-76.547,-176.130,8.183,148.477
C03558=1192.371,356.657,-76.514,-176.132,8.180,148.477
C03559=1192.375,356.409,-76.481,-176.134,8.177,148.476
C03560=1192.379,356.162,-76.447,-176.136,8.173,148.476
C03561=1192.383,355.914,-76.414,-176.138,8.170,148.476
C03562=1192.387,355.667,-76.380,-176.140,8.166,148.475
C03563=1192.391,355.419,-76.347,-176.142,8.163,148.475
C03564=1192.395,355.171,-76.314,-176.144,8.160,148.475
C03565=1192.399,354.923,-76.281,-176.146,8.157,148.475
C03566=1192.403,354.675,-76.247,-176.148,8.153,148.474
C03567=1192.407,354.427,-76.214,-176.150,8.150,148.474
C03568=1192.411,354.180,-76.181,-176.152,8.147,148.474
C03569=1192.415,353.932,-76.148,-176.154,8.143,148.473
C03570=1192.419,353.684,-76.115,-176.156,8.140,148.473
C03571=1192.424,353.436,-76.082,-176.158,8.137,148.473
C03572=1192.428,353.189,-76.048,-176.160,8.134,148.473
C03573=1192.432,352.941,-76.015,-176.162,8.130,148.472
C03574=1192.436,352.693,-75.982,-176.164,8.127,148.472
C03575=1192.440,352.446,-75.949,-176.166,8.124,148.472
C03576=1192.444,352.198,-75.916,-176.168,8.121,148.472
C03577=1192.448,351.950,-75.883,-176.170,8.117,148.471
C03578=1192.453,351.702,-75.850,-176.172,8.114,148.471
C03579=1192.457,351.455,-75.816,-176.174,8.111,148.471
C03580=1192.461,351.207,-75.783,-176.177,8.107,148.470
C03581=1192.465,350.959,-75.750,-176.178,8.105,148.470
C03582=1192.469,350.711,-75.717,-176.180,8.101,148.470
C03583=1192.473,350.464,-75.684,-176.182,8.098,148.470
C03584=1192.477,350.216,-75.651,-176.185,8.095,148.469
C03585=1192.482,349.968,-75.617,-176.187,8.091,148.469
C03586=1192.486,349.721,-75.584,-176.189,8.088,148.469
C03587=1192.489,349.473,-75.552,-176.191,8.085,148.469
C03588=1192.494,349.225,-75.519,-176.193,8.082,148.469
C03589=1192.498,348.977,-75.486,-176.195,8.079,148.468
C03590=1192.502,348.729,-75.453,-176.197,8.075,148.468
C03591=1192.506,348.482,-75.420,-176.199,8.072,148.468
C03592=1192.510,348.233,-75.387,-176.201,8.069,148.467
C03593=1192.515,347.986,-75.354,-176.203,8.066,148.467
C03594=1192.518,347.738,-75.322,-176.205,8.063,148.467
C03595=1192.522,347.490,-75.288,-176.208,8.059,148.467
C03596=1192.527,347.242,-75.256,-176.210,8.056,148.467
C03597=1192.531,346.994,-75.223,-176.212,8.053,148.466
C03598=1192.535,346.747,-75.190,-176.214,8.049,148.466
C03599=1192.539,346.498,-75.157,-176.216,8.047,148.466
C03600=1192.543,346.251,-75.125,-176.218,8.044,148.466
C03601=1192.547,346.003,-75.092,-176.221,8.040,148.466
C03602=1192.551,345.755,-75.059,-176.223,8.037,148.465
C03603=1192.555,345.507,-75.026,-176.225,8.034,148.465
C03604=1192.559,345.260,-74.994,-176.227,8.030,148.465
C03605=1192.564,345.012,-74.961,-176.229,8.028,148.465
C03606=1192.568,344.764,-74.928,-176.231,8.024,148.465
C03607=1192.572,344.516,-74.895,-176.233,8.021,148.464
C03608=1192.576,344.268,-74.863,-176.236,8.018,148.464
C03609=1192.580,344.021,-74.830,-176.238,8.014,148.464
C03610=1192.584,343.772,-74.798,-176.240,8.011,148.464
C03611=1192.589,343.525,-74.764,-176.242,8.009,148.464
C03612=1192.593,343.277,-74.733,-176.244,8.005,148.463
C03613=1192.597,343.030,-74.700,-176.246,8.002,148.463
C03614=1192.601,342.781,-74.667,-176.249,7.999,148.463
C03615=1192.605,342.534,-74.635,-176.251,7.995,148.463
C03616=1192.609,342.285,-74.602,-176.253,7.992,148.462
C03617=1192.613,342.038,-74.569,-176.255,7.990,148.462
C03618=1192.617,341.790,-74.537,-176.257,7.986,148.462
C03619=1192.622,341.543,-74.505,-176.260,7.983,148.462
C03620=1192.626,341.294,-74.472,-176.262,7.980,148.462
C03621=1192.630,341.047,-74.440,-176.264,7.977,148.462
C03622=1192.634,340.768,-74.404,-176.266,7.973,148.461
C03623=1192.640,340.489,-74.367,-176.269,7.970,148.461
C03624=1192.644,340.210,-74.330,-176.272,7.966,148.461
C03625=1192.649,339.932,-74.293,-176.274,7.963,148.461
C03626=1192.653,339.684,-74.262,-176.276,7.959,148.461
C03627=1192.657,339.436,-74.229,-176.279,7.956,148.460
C03628=1192.661,339.189,-74.197,-176.280,7.954,148.460
C03629=1192.665,338.940,-74.164,-176.282,7.950,148.460
C03630=1192.669,338.692,-74.133,-176.285,7.947,148.460
C03631=1192.674,338.445,-74.100,-176.287,7.944,148.460
C03632=1192.678,338.197,-74.067,-176.290,7.941,148.460
C03633=1192.682,337.949,-74.036,-176.292,7.937,148.459
C03634=1192.686,337.700,-74.003,-176.294,7.935,148.459
C03635=1192.690,337.454,-73.971,-176.296,7.932,148.459
C03636=1192.695,337.205,-73.939,-176.299,7.928,148.459
C03637=1192.698,336.957,-73.907,-176.301,7.925,148.459
C03638=1192.703,336.709,-73.874,-176.303,7.922,148.459
C03639=1192.707,336.462,-73.842,-176.305,7.920,148.459
C03640=1192.710,336.214,-73.810,-176.307,7.916,148.458
C03641=1192.715,335.966,-73.778,-176.310,7.913,148.458
C03642=1192.719,335.718,-73.746,-176.312,7.910,148.458
C03643=1192.724,335.470,-73.714,-176.315,7.907,148.458
C03644=1192.727,335.222,-73.682,-176.317,7.903,148.458
C03645=1192.732,334.974,-73.650,-176.319,7.901,148.458
C03646=1192.735,334.726,-73.617,-176.321,7.898,148.458
C03647=1192.740,334.479,-73.585,-176.323,7.894,148.457
C03648=1192.744,334.231,-73.553,-176.326,7.891,148.457
C03649=1192.748,333.983,-73.521,-176.328,7.888,148.457
C03650=1192.753,333.735,-73.489,-176.331,7.885,148.457
C03651=1192.756,333.487,-73.457,-176.332,7.882,148.457
C03652=1192.760,333.239,-73.425,-176.335,7.879,148.457
C03653=1192.765,332.991,-73.393,-176.337,7.876,148.457
C03654=1192.769,332.743,-73.362,-176.339,7.872,148.456
C03655=1192.773,332.495,-73.329,-176.342,7.869,148.456
C03656=1192.778,332.248,-73.298,-176.344,7.867,148.456
